SPLINE
SPL {X  -159.990, Y  +512.735, Z    +0.000, E1   +42.369, E3 +305939.523}
SPL {X  -159.990, Y  +505.924, Z    +0.000, E1   +43.199, E3 +305950.181}
SPL {X  -159.990, Y  +497.983, Z    +0.000, E1   +44.027, E3 +305963.054}
SPL {X  -159.990, Y  +489.703, Z    +0.000, E1   +44.938, E3 +305975.473}
SPL {X  -159.990, Y  +484.712, Z    +0.000, E1   +45.426, E3 +305983.087}
SPL {X  -159.990, Y  +477.648, Z    +0.000, E1   +46.080, E3 +305993.907}
SPL {X  -159.990, Y  +469.952, Z    +0.000, E1   +46.750, E3 +306005.415}
SPL {X  -159.990, Y  +462.892, Z    +0.000, E1   +47.497, E3 +306014.899}
SPL {X  -159.990, Y  +450.424, Z    +0.000, E1   +48.824, E3 +306030.863}
SPL {X  -159.990, Y  +436.919, Z    +0.000, E1   +49.944, E3 +306048.632}
SPL {X  -159.990, Y  +429.517, Z    +0.000, E1   +50.043, E3 +306061.146}
SPL {X  -159.990, Y  +423.834, Z    +0.000, E1   +50.037, E3 +306071.258}
SPL {X  -159.990, Y  +417.693, Z    +0.000, E1   +50.049, E3 +306082.156}
SPL {X  -159.990, Y  +408.922, Z    +0.000, E1   +50.085, E3 +306097.686}
SPL {X  -159.990, Y  +399.787, Z    +0.000, E1   +50.064, E3 +306113.955}
SPL {X  -159.990, Y  +393.038, Z    +0.000, E1   +50.038, E3 +306125.989}
SPL {X  -159.990, Y  +385.182, Z    +0.000, E1   +50.081, E3 +306139.906}
SPL {X  -159.906, Y  +377.302, Z    +0.000, E1   +50.024, E3 +306154.067}
SPL {X  -159.545, Y  +370.569, Z    +0.000, E1   +49.982, E3 +306166.380}
SPL {X  -158.871, Y  +363.614, Z    +0.000, E1   +49.855, E3 +306179.459}
SPL {X  -158.179, Y  +358.495, Z    +0.000, E1   +49.715, E3 +306189.308}
SPL {X  -157.354, Y  +353.576, Z    +0.000, E1   +49.583, E3 +306198.894}
SPL {X  -156.029, Y  +347.121, Z    +0.000, E1   +49.358, E3 +306211.711}
SPL {X  -154.686, Y  +341.646, Z    +0.000, E1   +49.094, E3 +306222.855}
SPL {X  -153.089, Y  +336.017, Z    +0.000, E1   +48.817, E3 +306234.464}
SPL {X  -151.481, Y  +331.019, Z    +0.000, E1   +48.491, E3 +306245.012}
SPL {X  -149.787, Y  +326.281, Z    +0.000, E1   +48.192, E3 +306255.100}
SPL {X  -148.124, Y  +322.035, Z    +0.000, E1   +47.846, E3 +306264.324}
SPL {X  -146.510, Y  +318.222, Z    +0.000, E1   +47.558, E3 +306272.636}
SPL {X  -141.189, Y  +307.250, Z    +0.000, E1   +40.067, E3 +306358.810}
ENDSPLINE

SPLINE
SPL {X  -154.923, Y  +342.556, Z    +0.000, E1   +23.930, E3 +306420.309}
SPL {X  -158.138, Y  +358.230, Z    +0.000, E1   +16.243, E3 +306429.267}
SPL {X  -159.647, Y  +372.034, Z    +0.000, E1    +8.739, E3 +306433.631}
SPL {X  -159.989, Y  +381.927, Z    +0.000, E1    +2.565, E3 +306435.391}
SPL {X  -159.990, Y  +386.909, Z    +0.000, E1    -1.211, E3 +306435.934}
SPL {X  -159.990, Y  +390.921, Z    +0.000, E1    -5.111, E3 +306436.413}
SPL {X  -159.990, Y  +395.719, Z    +0.000, E1   -10.396, E3 +306437.232}
SPL {X  -159.990, Y  +400.739, Z    +0.000, E1   -16.236, E3 +306438.430}
SPL {X  -159.990, Y  +409.482, Z    +0.000, E1   -25.418, E3 +306441.635}
SPL {X  -159.990, Y  +440.741, Z    +0.000, E1   -43.570, E3 +306462.292}
SPL {X  -159.990, Y  +489.732, Z    +0.000, E1   -48.863, E3 +306526.450}
SPL {X  -159.990, Y  +496.901, Z    +0.000, E1   -48.832, E3 +306539.797}
SPL {X  -159.990, Y  +502.531, Z    +0.000, E1   -48.834, E3 +306550.242}
SPL {X  -159.990, Y  +508.013, Z    +0.000, E1   -48.835, E3 +306560.377}
SPL {X  -159.990, Y  +513.813, Z    +0.000, E1   -48.843, E3 +306571.125}
SPL {X  -159.990, Y  +522.177, Z    +0.000, E1   -48.881, E3 +306586.602}
SPL {X  -159.990, Y  +532.076, Z    +0.000, E1   -48.872, E3 +306604.975}
SPL {X  -159.990, Y  +539.248, Z    +0.000, E1   -48.832, E3 +306618.343}
SPL {X  -159.990, Y  +544.926, Z    +0.000, E1   -48.835, E3 +306628.872}
SPL {X  -159.990, Y  +550.252, Z    +0.000, E1   -48.827, E3 +306638.778}
SPL {X  -159.990, Y  +555.692, Z    +0.000, E1   -48.830, E3 +306648.875}
SPL {X  -159.990, Y  +561.308, Z    +0.000, E1   -48.827, E3 +306659.322}
SPL {X  -159.990, Y  +566.669, Z    +0.000, E1   -48.820, E3 +306669.271}
SPL {X  -159.990, Y  +572.248, Z    +0.000, E1   -48.830, E3 +306679.616}
SPL {X  -159.990, Y  +577.770, Z    +0.000, E1   -48.821, E3 +306689.863}
SPL {X  -159.990, Y  +583.108, Z    +0.000, E1   -48.828, E3 +306699.765}
SPL {X  -159.990, Y  +588.804, Z    +0.000, E1   -48.829, E3 +306710.322}
SPL {X  -159.990, Y  +594.280, Z    +0.000, E1   -48.826, E3 +306720.484}
SPL {X  -159.990, Y  +600.107, Z    +0.000, E1   -48.833, E3 +306731.298}
SPL {X  -159.990, Y  +605.910, Z    +0.000, E1   -48.823, E3 +306742.077}
SPL {X  -159.990, Y  +611.566, Z    +0.000, E1   -48.829, E3 +306752.566}
SPL {X  -159.990, Y  +617.357, Z    +0.000, E1   -48.824, E3 +306763.321}
SPL {X  -159.990, Y  +622.965, Z    +0.000, E1   -48.826, E3 +306773.720}
SPL {X  -159.990, Y  +629.255, Z    +0.000, E1   -48.834, E3 +306785.387}
SPL {X  -159.990, Y  +634.905, Z    +0.000, E1   -48.821, E3 +306795.884}
SPL {X  -159.990, Y  +640.372, Z    +0.000, E1   -48.828, E3 +306806.021}
SPL {X  -159.990, Y  +646.939, Z    +0.000, E1   -48.838, E3 +306818.191}
SPL {X  -159.990, Y  +653.448, Z    +0.000, E1   -48.827, E3 +306830.286}
SPL {X  -159.990, Y  +659.039, Z    +0.000, E1   -48.826, E3 +306840.650}
SPL {X  -159.990, Y  +664.817, Z    +0.000, E1   -48.832, E3 +306851.365}
SPL {X  -159.990, Y  +671.221, Z    +0.000, E1   -48.836, E3 +306863.238}
SPL {X  -159.887, Y  +677.230, Z    +0.000, E1   -48.811, E3 +306874.504}
SPL {X  -159.602, Y  +682.629, Z    +0.000, E1   -48.761, E3 +306884.837}
SPL {X  -159.150, Y  +687.876, Z    +0.000, E1   -48.673, E3 +306895.076}
SPL {X  -158.569, Y  +692.776, Z    +0.000, E1   -48.570, E3 +306904.784}
SPL {X  -157.870, Y  +697.458, Z    +0.000, E1   -48.439, E3 +306914.213}
SPL {X  -157.028, Y  +702.144, Z    +0.000, E1   -48.297, E3 +306923.761}
SPL {X  -155.977, Y  +707.110, Z    +0.000, E1   -48.106, E3 +306934.065}
SPL {X  -154.657, Y  +712.464, Z    +0.000, E1   -47.874, E3 +306945.349}
SPL {X  -153.406, Y  +716.924, Z    +0.000, E1   -47.628, E3 +306954.915}
SPL {X  -152.020, Y  +721.367, Z    +0.000, E1   -47.374, E3 +306964.566}
SPL {X  -150.440, Y  +725.947, Z    +0.000, E1   -47.070, E3 +306974.671}
SPL {X  -148.730, Y  +730.459, Z    +0.000, E1   -46.749, E3 +306984.722}
SPL {X  -147.178, Y  +734.233, Z    +0.000, E1   -46.439, E3 +306993.256}
SPL {X  -140.222, Y  +748.536, Z    +0.000, E1   -42.074, E3 +307058.232}
ENDSPLINE

SPLINE
SPL {X  -152.021, Y  +721.365, Z    +0.000, E1   -28.339, E3 +307133.623}
SPL {X  -157.542, Y  +699.382, Z    +0.000, E1   -18.086, E3 +307149.141}
SPL {X  -159.386, Y  +685.393, Z    +0.000, E1   -10.664, E3 +307154.095}
SPL {X  -159.928, Y  +675.946, Z    +0.000, E1    -5.007, E3 +307156.134}
SPL {X  -159.990, Y  +671.468, Z    +0.000, E1    -2.030, E3 +307156.730}
SPL {X  -159.990, Y  +667.678, Z    +0.000, E1    +0.783, E3 +307157.080}
SPL {X  -159.990, Y  +663.139, Z    +0.000, E1    +5.135, E3 +307157.597}
SPL {X  -159.990, Y  +658.551, Z    +0.000, E1   +10.313, E3 +307158.371}
SPL {X  -159.990, Y  +653.526, Z    +0.000, E1   +16.156, E3 +307159.606}
SPL {X  -159.990, Y  +644.434, Z    +0.000, E1   +25.921, E3 +307162.801}
SPL {X  -159.990, Y  +612.255, Z    +0.000, E1   +44.102, E3 +307184.682}
SPL {X  -159.990, Y  +562.879, Z    +0.000, E1   +49.634, E3 +307246.271}
SPL {X  -159.990, Y  +554.544, Z    +0.000, E1   +49.649, E3 +307261.296}
SPL {X  -159.990, Y  +547.278, Z    +0.000, E1   +49.619, E3 +307274.455}
SPL {X  -159.990, Y  +540.489, Z    +0.000, E1   +49.634, E3 +307286.681}
SPL {X  -159.990, Y  +532.689, Z    +0.000, E1   +49.639, E3 +307300.734}
SPL {X  -159.990, Y  +524.316, Z    +0.000, E1   +49.648, E3 +307315.819}
SPL {X  -159.990, Y  +517.666, Z    +0.000, E1   +49.614, E3 +307327.880}
SPL {X  -159.990, Y  +511.038, Z    +0.000, E1   +49.636, E3 +307339.832}
SPL {X  -159.990, Y  +504.260, Z    +0.000, E1   +49.614, E3 +307352.105}
ENDSPLINE

SPLINE
SPL {X  -159.990, Y  +511.561, Z    +0.000, E1   +45.946, E3 +307359.627}
SPL {X  -159.990, Y  +518.175, Z    +0.000, E1   +41.708, E3 +307370.702}
ENDSPLINE

SPLINE
SPL {X  -159.990, Y  +508.096, Z    +0.000, E1   +42.952, E3 +307386.810}
SPL {X  -159.990, Y  +497.983, Z    +0.000, E1   +44.027, E3 +307403.054}
SPL {X  -159.990, Y  +489.703, Z    +0.000, E1   +44.938, E3 +307415.473}
SPL {X  -159.990, Y  +482.131, Z    +0.000, E1   +45.680, E3 +307427.053}
SPL {X  -159.990, Y  +472.111, Z    +0.000, E1   +46.581, E3 +307442.185}
SPL {X  -159.990, Y  +462.892, Z    +0.000, E1   +47.497, E3 +307454.899}
SPL {X  -159.990, Y  +452.841, Z    +0.000, E1   +48.572, E3 +307467.746}
SPL {X  -159.990, Y  +441.023, Z    +0.000, E1   +49.655, E3 +307482.997}
SPL {X  -159.990, Y  +431.096, Z    +0.000, E1   +50.075, E3 +307498.285}
SPL {X  -159.990, Y  +421.718, Z    +0.000, E1   +50.072, E3 +307514.965}
SPL {X  -159.990, Y  +412.896, Z    +0.000, E1   +50.065, E3 +307530.658}
SPL {X  -159.990, Y  +406.170, Z    +0.000, E1   +50.036, E3 +307542.647}
SPL {X  -159.990, Y  +399.787, Z    +0.000, E1   +50.064, E3 +307553.955}
SPL {X  -159.990, Y  +393.038, Z    +0.000, E1   +50.038, E3 +307565.989}
SPL {X  -159.990, Y  +385.182, Z    +0.000, E1   +50.081, E3 +307579.906}
SPL {X  -159.846, Y  +375.718, Z    +0.000, E1   +50.041, E3 +307596.901}
SPL {X  -159.300, Y  +367.653, Z    +0.000, E1   +49.944, E3 +307611.809}
SPL {X  -158.412, Y  +360.086, Z    +0.000, E1   +49.787, E3 +307626.191}
SPL {X  -157.354, Y  +353.576, Z    +0.000, E1   +49.583, E3 +307638.894}
SPL {X  -156.029, Y  +347.121, Z    +0.000, E1   +49.358, E3 +307651.711}
SPL {X  -154.686, Y  +341.646, Z    +0.000, E1   +49.094, E3 +307662.855}
SPL {X  -153.089, Y  +336.017, Z    +0.000, E1   +48.817, E3 +307674.464}
SPL {X  -151.481, Y  +331.019, Z    +0.000, E1   +48.491, E3 +307685.012}
SPL {X  -150.221, Y  +327.451, Z    +0.000, E1   +48.251, E3 +307692.616}
SPL {X  -148.587, Y  +323.181, Z    +0.000, E1   +47.960, E3 +307701.800}
SPL {X  -146.510, Y  +318.222, Z    +0.000, E1   +47.558, E3 +307712.636}
SPL {X  -141.189, Y  +307.250, Z    +0.000, E1   +40.067, E3 +307798.810}
ENDSPLINE

SPLINE
SPL {X  -154.923, Y  +342.556, Z    +0.000, E1   +23.930, E3 +307860.309}
SPL {X  -158.138, Y  +358.230, Z    +0.000, E1   +16.243, E3 +307869.267}
SPL {X  -159.647, Y  +372.034, Z    +0.000, E1    +8.739, E3 +307873.631}
SPL {X  -159.989, Y  +381.927, Z    +0.000, E1    +2.565, E3 +307875.391}
SPL {X  -159.990, Y  +386.909, Z    +0.000, E1    -1.211, E3 +307875.934}
SPL {X  -159.990, Y  +390.921, Z    +0.000, E1    -5.111, E3 +307876.413}
SPL {X  -159.990, Y  +395.719, Z    +0.000, E1   -10.396, E3 +307877.232}
SPL {X  -159.990, Y  +400.739, Z    +0.000, E1   -16.236, E3 +307878.430}
SPL {X  -159.990, Y  +409.482, Z    +0.000, E1   -25.418, E3 +307881.635}
SPL {X  -159.990, Y  +440.741, Z    +0.000, E1   -43.570, E3 +307902.292}
SPL {X  -159.990, Y  +488.072, Z    +0.000, E1   -48.834, E3 +307963.414}
SPL {X  -159.990, Y  +495.397, Z    +0.000, E1   -48.860, E3 +307976.963}
SPL {X  -159.990, Y  +502.531, Z    +0.000, E1   -48.834, E3 +307990.242}
SPL {X  -159.990, Y  +508.013, Z    +0.000, E1   -48.835, E3 +308000.377}
SPL {X  -159.990, Y  +513.813, Z    +0.000, E1   -48.843, E3 +308011.125}
SPL {X  -159.990, Y  +522.177, Z    +0.000, E1   -48.881, E3 +308026.602}
SPL {X  -159.990, Y  +532.076, Z    +0.000, E1   -48.872, E3 +308044.975}
SPL {X  -159.990, Y  +539.248, Z    +0.000, E1   -48.832, E3 +308058.343}
SPL {X  -159.990, Y  +544.926, Z    +0.000, E1   -48.835, E3 +308068.872}
SPL {X  -159.990, Y  +550.252, Z    +0.000, E1   -48.827, E3 +308078.778}
SPL {X  -159.990, Y  +555.692, Z    +0.000, E1   -48.830, E3 +308088.875}
SPL {X  -159.990, Y  +561.308, Z    +0.000, E1   -48.827, E3 +308099.322}
SPL {X  -159.990, Y  +566.669, Z    +0.000, E1   -48.820, E3 +308109.271}
SPL {X  -159.990, Y  +572.248, Z    +0.000, E1   -48.830, E3 +308119.616}
SPL {X  -159.990, Y  +577.770, Z    +0.000, E1   -48.821, E3 +308129.863}
SPL {X  -159.990, Y  +583.108, Z    +0.000, E1   -48.828, E3 +308139.765}
SPL {X  -159.990, Y  +588.804, Z    +0.000, E1   -48.829, E3 +308150.322}
SPL {X  -159.990, Y  +594.280, Z    +0.000, E1   -48.826, E3 +308160.484}
SPL {X  -159.990, Y  +600.107, Z    +0.000, E1   -48.833, E3 +308171.298}
SPL {X  -159.990, Y  +605.910, Z    +0.000, E1   -48.823, E3 +308182.077}
SPL {X  -159.990, Y  +611.566, Z    +0.000, E1   -48.829, E3 +308192.566}
SPL {X  -159.990, Y  +617.357, Z    +0.000, E1   -48.824, E3 +308203.321}
SPL {X  -159.990, Y  +622.965, Z    +0.000, E1   -48.826, E3 +308213.720}
SPL {X  -159.990, Y  +629.255, Z    +0.000, E1   -48.834, E3 +308225.387}
SPL {X  -159.990, Y  +634.905, Z    +0.000, E1   -48.821, E3 +308235.884}
SPL {X  -159.990, Y  +640.372, Z    +0.000, E1   -48.828, E3 +308246.021}
SPL {X  -159.990, Y  +646.939, Z    +0.000, E1   -48.838, E3 +308258.191}
SPL {X  -159.990, Y  +653.448, Z    +0.000, E1   -48.827, E3 +308270.286}
SPL {X  -159.990, Y  +659.039, Z    +0.000, E1   -48.826, E3 +308280.650}
SPL {X  -159.990, Y  +664.817, Z    +0.000, E1   -48.832, E3 +308291.365}
SPL {X  -159.990, Y  +671.221, Z    +0.000, E1   -48.836, E3 +308303.238}
SPL {X  -159.887, Y  +677.230, Z    +0.000, E1   -48.811, E3 +308314.504}
SPL {X  -159.602, Y  +682.629, Z    +0.000, E1   -48.761, E3 +308324.837}
SPL {X  -159.150, Y  +687.876, Z    +0.000, E1   -48.673, E3 +308335.076}
SPL {X  -158.569, Y  +692.776, Z    +0.000, E1   -48.570, E3 +308344.784}
SPL {X  -157.870, Y  +697.458, Z    +0.000, E1   -48.439, E3 +308354.213}
SPL {X  -157.028, Y  +702.144, Z    +0.000, E1   -48.297, E3 +308363.761}
SPL {X  -155.977, Y  +707.110, Z    +0.000, E1   -48.106, E3 +308374.065}
SPL {X  -154.657, Y  +712.464, Z    +0.000, E1   -47.874, E3 +308385.349}
SPL {X  -153.406, Y  +716.924, Z    +0.000, E1   -47.628, E3 +308394.915}
SPL {X  -152.020, Y  +721.367, Z    +0.000, E1   -47.374, E3 +308404.566}
SPL {X  -150.440, Y  +725.947, Z    +0.000, E1   -47.070, E3 +308414.671}
SPL {X  -148.730, Y  +730.459, Z    +0.000, E1   -46.749, E3 +308424.722}
SPL {X  -147.178, Y  +734.233, Z    +0.000, E1   -46.439, E3 +308433.256}
SPL {X  -140.263, Y  +748.461, Z    +0.000, E1   -42.675, E3 +308491.594}
ENDSPLINE

SPLINE
SPL {X  -141.835, Y  +745.525, Z    +0.000, E1   -39.068, E3 +308523.595}
SPL {X  -152.406, Y  +720.176, Z    +0.000, E1   -27.814, E3 +308574.808}
SPL {X  -158.165, Y  +695.595, Z    +0.000, E1   -16.189, E3 +308590.706}
SPL {X  -159.572, Y  +683.063, Z    +0.000, E1    -9.282, E3 +308594.713}
SPL {X  -159.928, Y  +675.946, Z    +0.000, E1    -5.007, E3 +308596.134}
SPL {X  -159.990, Y  +671.468, Z    +0.000, E1    -2.030, E3 +308596.730}
SPL {X  -159.990, Y  +667.678, Z    +0.000, E1    +0.783, E3 +308597.080}
SPL {X  -159.990, Y  +663.139, Z    +0.000, E1    +5.135, E3 +308597.597}
SPL {X  -159.990, Y  +658.551, Z    +0.000, E1   +10.313, E3 +308598.371}
SPL {X  -159.990, Y  +653.526, Z    +0.000, E1   +16.156, E3 +308599.606}
SPL {X  -159.990, Y  +644.434, Z    +0.000, E1   +25.921, E3 +308602.801}
SPL {X  -159.990, Y  +612.255, Z    +0.000, E1   +44.102, E3 +308624.682}
SPL {X  -159.990, Y  +567.037, Z    +0.000, E1   +49.607, E3 +308678.826}
SPL {X  -159.990, Y  +562.169, Z    +0.000, E1   +49.620, E3 +308687.582}
SPL {X  -159.990, Y  +554.544, Z    +0.000, E1   +49.649, E3 +308701.296}
SPL {X  -159.990, Y  +545.715, Z    +0.000, E1   +49.644, E3 +308717.240}
SPL {X  -159.990, Y  +537.339, Z    +0.000, E1   +49.638, E3 +308732.351}
SPL {X  -159.990, Y  +529.436, Z    +0.000, E1   +49.638, E3 +308746.603}
SPL {X  -159.990, Y  +520.280, Z    +0.000, E1   +49.665, E3 +308763.082}
SPL {X  -159.990, Y  +511.038, Z    +0.000, E1   +49.636, E3 +308779.832}
SPL {X  -159.990, Y  +504.260, Z    +0.000, E1   +49.614, E3 +308792.105}
ENDSPLINE

SPLINE
SPL {X  -159.990, Y  +511.561, Z    +0.000, E1   +45.946, E3 +308799.627}
SPL {X  -159.990, Y  +518.175, Z    +0.000, E1   +41.708, E3 +308810.702}
ENDSPLINE

SPLINE
SPL {X  -159.990, Y  +508.096, Z    +0.000, E1   +42.952, E3 +308826.810}
SPL {X  -159.990, Y  +497.983, Z    +0.000, E1   +44.027, E3 +308843.054}
SPL {X  -159.990, Y  +487.435, Z    +0.000, E1   +45.185, E3 +308858.910}
SPL {X  -159.990, Y  +477.648, Z    +0.000, E1   +46.080, E3 +308873.907}
SPL {X  -159.990, Y  +469.952, Z    +0.000, E1   +46.750, E3 +308885.415}
SPL {X  -159.990, Y  +462.892, Z    +0.000, E1   +47.497, E3 +308894.899}
SPL {X  -159.990, Y  +452.841, Z    +0.000, E1   +48.572, E3 +308907.746}
SPL {X  -159.990, Y  +439.038, Z    +0.000, E1   +49.804, E3 +308925.798}
SPL {X  -159.990, Y  +429.517, Z    +0.000, E1   +50.043, E3 +308941.146}
SPL {X  -159.990, Y  +423.834, Z    +0.000, E1   +50.037, E3 +308951.258}
SPL {X  -159.990, Y  +417.693, Z    +0.000, E1   +50.049, E3 +308962.156}
SPL {X  -159.990, Y  +411.447, Z    +0.000, E1   +50.039, E3 +308973.275}
SPL {X  -159.990, Y  +403.654, Z    +0.000, E1   +50.076, E3 +308987.065}
SPL {X  -159.990, Y  +394.612, Z    +0.000, E1   +50.064, E3 +309003.153}
SPL {X  -159.990, Y  +385.182, Z    +0.000, E1   +50.081, E3 +309019.906}
SPL {X  -159.846, Y  +375.718, Z    +0.000, E1   +50.041, E3 +309036.901}
SPL {X  -159.300, Y  +367.653, Z    +0.000, E1   +49.944, E3 +309051.809}
SPL {X  -158.412, Y  +360.086, Z    +0.000, E1   +49.787, E3 +309066.191}
SPL {X  -157.077, Y  +352.107, Z    +0.000, E1   +49.567, E3 +309081.742}
SPL {X  -155.744, Y  +345.884, Z    +0.000, E1   +49.283, E3 +309094.229}
SPL {X  -154.686, Y  +341.646, Z    +0.000, E1   +49.094, E3 +309102.855}
SPL {X  -153.089, Y  +336.017, Z    +0.000, E1   +48.817, E3 +309114.464}
SPL {X  -150.861, Y  +329.230, Z    +0.000, E1   +48.419, E3 +309128.753}
SPL {X  -148.587, Y  +323.181, Z    +0.000, E1   +47.960, E3 +309141.800}
SPL {X  -146.885, Y  +319.085, Z    +0.000, E1   +47.613, E3 +309150.761}
SPL {X  -145.797, Y  +316.621, Z    +0.000, E1   +47.387, E3 +309156.210}
SPL {X  -141.189, Y  +307.250, Z    +0.000, E1   +40.067, E3 +309238.810}
ENDSPLINE

SPLINE
SPL {X  -154.923, Y  +342.556, Z    +0.000, E1   +23.930, E3 +309300.309}
SPL {X  -158.138, Y  +358.230, Z    +0.000, E1   +16.243, E3 +309309.267}
SPL {X  -159.407, Y  +368.849, Z    +0.000, E1   +10.504, E3 +309312.867}
SPL {X  -159.931, Y  +378.162, Z    +0.000, E1    +5.020, E3 +309314.852}
SPL {X  -159.990, Y  +383.297, Z    +0.000, E1    +1.526, E3 +309315.557}
SPL {X  -159.990, Y  +386.909, Z    +0.000, E1    -1.211, E3 +309315.934}
SPL {X  -159.990, Y  +390.921, Z    +0.000, E1    -5.111, E3 +309316.413}
SPL {X  -159.990, Y  +395.719, Z    +0.000, E1   -10.396, E3 +309317.232}
SPL {X  -159.990, Y  +400.739, Z    +0.000, E1   -16.236, E3 +309318.430}
SPL {X  -159.990, Y  +409.482, Z    +0.000, E1   -25.418, E3 +309321.635}
SPL {X  -159.990, Y  +440.741, Z    +0.000, E1   -43.570, E3 +309342.292}
SPL {X  -159.990, Y  +489.732, Z    +0.000, E1   -48.863, E3 +309406.450}
SPL {X  -159.990, Y  +496.901, Z    +0.000, E1   -48.832, E3 +309419.797}
SPL {X  -159.990, Y  +502.531, Z    +0.000, E1   -48.834, E3 +309430.242}
SPL {X  -159.990, Y  +508.013, Z    +0.000, E1   -48.835, E3 +309440.377}
SPL {X  -159.990, Y  +513.813, Z    +0.000, E1   -48.843, E3 +309451.125}
SPL {X  -159.990, Y  +522.177, Z    +0.000, E1   -48.881, E3 +309466.602}
SPL {X  -159.990, Y  +532.076, Z    +0.000, E1   -48.872, E3 +309484.975}
SPL {X  -159.990, Y  +539.248, Z    +0.000, E1   -48.832, E3 +309498.343}
SPL {X  -159.990, Y  +544.926, Z    +0.000, E1   -48.835, E3 +309508.872}
SPL {X  -159.990, Y  +550.252, Z    +0.000, E1   -48.827, E3 +309518.778}
SPL {X  -159.990, Y  +555.692, Z    +0.000, E1   -48.830, E3 +309528.875}
SPL {X  -159.990, Y  +561.308, Z    +0.000, E1   -48.827, E3 +309539.322}
SPL {X  -159.990, Y  +566.669, Z    +0.000, E1   -48.820, E3 +309549.271}
SPL {X  -159.990, Y  +572.248, Z    +0.000, E1   -48.830, E3 +309559.616}
SPL {X  -159.990, Y  +577.770, Z    +0.000, E1   -48.821, E3 +309569.863}
SPL {X  -159.990, Y  +583.108, Z    +0.000, E1   -48.828, E3 +309579.765}
SPL {X  -159.990, Y  +588.804, Z    +0.000, E1   -48.829, E3 +309590.322}
SPL {X  -159.990, Y  +594.280, Z    +0.000, E1   -48.826, E3 +309600.484}
SPL {X  -159.990, Y  +600.107, Z    +0.000, E1   -48.833, E3 +309611.298}
SPL {X  -159.990, Y  +605.910, Z    +0.000, E1   -48.823, E3 +309622.077}
SPL {X  -159.990, Y  +611.566, Z    +0.000, E1   -48.829, E3 +309632.566}
SPL {X  -159.990, Y  +617.357, Z    +0.000, E1   -48.824, E3 +309643.321}
SPL {X  -159.990, Y  +622.965, Z    +0.000, E1   -48.826, E3 +309653.720}
SPL {X  -159.990, Y  +629.255, Z    +0.000, E1   -48.834, E3 +309665.387}
SPL {X  -159.990, Y  +634.905, Z    +0.000, E1   -48.821, E3 +309675.884}
SPL {X  -159.990, Y  +640.372, Z    +0.000, E1   -48.828, E3 +309686.021}
SPL {X  -159.990, Y  +646.939, Z    +0.000, E1   -48.838, E3 +309698.191}
SPL {X  -159.990, Y  +653.448, Z    +0.000, E1   -48.827, E3 +309710.286}
SPL {X  -159.990, Y  +659.039, Z    +0.000, E1   -48.826, E3 +309720.650}
SPL {X  -159.990, Y  +664.817, Z    +0.000, E1   -48.832, E3 +309731.365}
SPL {X  -159.990, Y  +671.221, Z    +0.000, E1   -48.836, E3 +309743.238}
SPL {X  -159.887, Y  +677.230, Z    +0.000, E1   -48.811, E3 +309754.504}
SPL {X  -159.602, Y  +682.629, Z    +0.000, E1   -48.761, E3 +309764.837}
SPL {X  -159.150, Y  +687.876, Z    +0.000, E1   -48.673, E3 +309775.076}
SPL {X  -158.569, Y  +692.776, Z    +0.000, E1   -48.570, E3 +309784.784}
SPL {X  -157.870, Y  +697.458, Z    +0.000, E1   -48.439, E3 +309794.213}
SPL {X  -157.028, Y  +702.144, Z    +0.000, E1   -48.297, E3 +309803.761}
SPL {X  -155.977, Y  +707.110, Z    +0.000, E1   -48.106, E3 +309814.065}
SPL {X  -154.657, Y  +712.464, Z    +0.000, E1   -47.874, E3 +309825.349}
SPL {X  -153.406, Y  +716.924, Z    +0.000, E1   -47.628, E3 +309834.915}
SPL {X  -152.020, Y  +721.367, Z    +0.000, E1   -47.374, E3 +309844.566}
SPL {X  -150.440, Y  +725.947, Z    +0.000, E1   -47.070, E3 +309854.671}
SPL {X  -148.730, Y  +730.459, Z    +0.000, E1   -46.749, E3 +309864.722}
SPL {X  -147.178, Y  +734.233, Z    +0.000, E1   -46.439, E3 +309873.256}
SPL {X  -140.222, Y  +748.536, Z    +0.000, E1   -42.074, E3 +309938.232}
ENDSPLINE

SPLINE
SPL {X  -152.021, Y  +721.365, Z    +0.000, E1   -28.339, E3 +310013.623}
SPL {X  -158.165, Y  +695.595, Z    +0.000, E1   -16.189, E3 +310030.706}
SPL {X  -159.572, Y  +683.063, Z    +0.000, E1    -9.282, E3 +310034.713}
SPL {X  -159.928, Y  +675.946, Z    +0.000, E1    -5.007, E3 +310036.134}
SPL {X  -159.990, Y  +669.697, Z    +0.000, E1    -0.851, E3 +310036.894}
SPL {X  -159.990, Y  +665.698, Z    +0.000, E1    +2.616, E3 +310037.273}
SPL {X  -159.990, Y  +662.251, Z    +0.000, E1    +6.155, E3 +310037.719}
SPL {X  -159.990, Y  +658.551, Z    +0.000, E1   +10.313, E3 +310038.371}
SPL {X  -159.990, Y  +653.526, Z    +0.000, E1   +16.156, E3 +310039.606}
SPL {X  -159.990, Y  +644.434, Z    +0.000, E1   +25.921, E3 +310042.801}
SPL {X  -159.990, Y  +612.255, Z    +0.000, E1   +44.102, E3 +310064.682}
SPL {X  -159.990, Y  +561.053, Z    +0.000, E1   +49.668, E3 +310129.515}
SPL {X  -159.990, Y  +552.984, Z    +0.000, E1   +49.619, E3 +310144.156}
SPL {X  -159.990, Y  +547.278, Z    +0.000, E1   +49.619, E3 +310154.455}
SPL {X  -159.990, Y  +538.738, Z    +0.000, E1   +49.672, E3 +310169.779}
SPL {X  -159.990, Y  +529.436, Z    +0.000, E1   +49.638, E3 +310186.603}
SPL {X  -159.990, Y  +522.804, Z    +0.000, E1   +49.620, E3 +310198.592}
SPL {X  -159.990, Y  +515.173, Z    +0.000, E1   +49.653, E3 +310212.330}
SPL {X  -159.990, Y  +505.472, Z    +0.000, E1   +49.465, E3 +310231.135}
ENDSPLINE

SPLINE
SPL {X  -159.990, Y  +518.841, Z    +0.000, E1   +41.643, E3 +310249.543}
ENDSPLINE

SPLINE
SPL {X  -159.990, Y  +508.096, Z    +0.000, E1   +42.952, E3 +310266.810}
SPL {X  -159.990, Y  +500.642, Z    +0.000, E1   +43.747, E3 +310278.731}
SPL {X  -159.990, Y  +495.820, Z    +0.000, E1   +44.207, E3 +310286.618}
SPL {X  -159.990, Y  +487.435, Z    +0.000, E1   +45.185, E3 +310298.910}
SPL {X  -159.990, Y  +477.648, Z    +0.000, E1   +46.080, E3 +310313.907}
SPL {X  -159.990, Y  +469.952, Z    +0.000, E1   +46.750, E3 +310325.415}
SPL {X  -159.990, Y  +462.892, Z    +0.000, E1   +47.497, E3 +310334.899}
SPL {X  -159.990, Y  +452.841, Z    +0.000, E1   +48.572, E3 +310347.746}
SPL {X  -159.990, Y  +439.038, Z    +0.000, E1   +49.804, E3 +310365.798}
SPL {X  -159.990, Y  +429.517, Z    +0.000, E1   +50.043, E3 +310381.146}
SPL {X  -159.990, Y  +423.834, Z    +0.000, E1   +50.037, E3 +310391.258}
SPL {X  -159.990, Y  +417.693, Z    +0.000, E1   +50.049, E3 +310402.156}
SPL {X  -159.990, Y  +411.447, Z    +0.000, E1   +50.039, E3 +310413.275}
SPL {X  -159.990, Y  +406.170, Z    +0.000, E1   +50.036, E3 +310422.647}
SPL {X  -159.990, Y  +399.787, Z    +0.000, E1   +50.064, E3 +310433.955}
SPL {X  -159.990, Y  +393.038, Z    +0.000, E1   +50.038, E3 +310445.989}
SPL {X  -159.990, Y  +387.356, Z    +0.000, E1   +50.042, E3 +310456.100}
SPL {X  -159.990, Y  +382.225, Z    +0.000, E1   +50.028, E3 +310465.245}
SPL {X  -159.846, Y  +375.718, Z    +0.000, E1   +50.041, E3 +310476.901}
SPL {X  -159.443, Y  +369.277, Z    +0.000, E1   +49.941, E3 +310488.815}
SPL {X  -158.871, Y  +363.614, Z    +0.000, E1   +49.855, E3 +310499.459}
SPL {X  -158.179, Y  +358.495, Z    +0.000, E1   +49.715, E3 +310509.308}
SPL {X  -157.077, Y  +352.107, Z    +0.000, E1   +49.567, E3 +310521.742}
SPL {X  -155.744, Y  +345.884, Z    +0.000, E1   +49.283, E3 +310534.229}
SPL {X  -154.686, Y  +341.646, Z    +0.000, E1   +49.094, E3 +310542.855}
SPL {X  -153.439, Y  +337.188, Z    +0.000, E1   +48.857, E3 +310552.062}
SPL {X  -151.836, Y  +332.074, Z    +0.000, E1   +48.585, E3 +310562.738}
SPL {X  -150.221, Y  +327.451, Z    +0.000, E1   +48.251, E3 +310572.616}
SPL {X  -148.587, Y  +323.181, Z    +0.000, E1   +47.960, E3 +310581.800}
SPL {X  -146.510, Y  +318.222, Z    +0.000, E1   +47.558, E3 +310592.636}
SPL {X  -141.189, Y  +307.250, Z    +0.000, E1   +40.067, E3 +310678.810}
ENDSPLINE

SPLINE
SPL {X  -154.923, Y  +342.556, Z    +0.000, E1   +23.930, E3 +310740.309}
SPL {X  -158.138, Y  +358.230, Z    +0.000, E1   +16.243, E3 +310749.267}
SPL {X  -159.647, Y  +372.034, Z    +0.000, E1    +8.739, E3 +310753.631}
SPL {X  -159.989, Y  +381.927, Z    +0.000, E1    +2.565, E3 +310755.391}
SPL {X  -159.990, Y  +386.909, Z    +0.000, E1    -1.211, E3 +310755.934}
SPL {X  -159.990, Y  +390.921, Z    +0.000, E1    -5.111, E3 +310756.413}
SPL {X  -159.990, Y  +395.719, Z    +0.000, E1   -10.396, E3 +310757.232}
SPL {X  -159.990, Y  +400.739, Z    +0.000, E1   -16.236, E3 +310758.430}
SPL {X  -159.990, Y  +409.482, Z    +0.000, E1   -25.418, E3 +310761.635}
SPL {X  -159.990, Y  +440.741, Z    +0.000, E1   -43.570, E3 +310782.292}
SPL {X  -159.990, Y  +489.732, Z    +0.000, E1   -48.863, E3 +310846.450}
SPL {X  -159.990, Y  +496.901, Z    +0.000, E1   -48.832, E3 +310859.797}
SPL {X  -159.990, Y  +502.531, Z    +0.000, E1   -48.834, E3 +310870.242}
SPL {X  -159.990, Y  +508.013, Z    +0.000, E1   -48.835, E3 +310880.377}
SPL {X  -159.990, Y  +513.813, Z    +0.000, E1   -48.843, E3 +310891.125}
SPL {X  -159.990, Y  +522.177, Z    +0.000, E1   -48.881, E3 +310906.602}
SPL {X  -159.990, Y  +532.076, Z    +0.000, E1   -48.872, E3 +310924.975}
SPL {X  -159.990, Y  +539.248, Z    +0.000, E1   -48.832, E3 +310938.343}
SPL {X  -159.990, Y  +544.926, Z    +0.000, E1   -48.835, E3 +310948.872}
SPL {X  -159.990, Y  +550.252, Z    +0.000, E1   -48.827, E3 +310958.778}
SPL {X  -159.990, Y  +555.692, Z    +0.000, E1   -48.830, E3 +310968.875}
SPL {X  -159.990, Y  +561.308, Z    +0.000, E1   -48.827, E3 +310979.322}
SPL {X  -159.990, Y  +566.669, Z    +0.000, E1   -48.820, E3 +310989.271}
SPL {X  -159.990, Y  +572.248, Z    +0.000, E1   -48.830, E3 +310999.616}
SPL {X  -159.990, Y  +577.770, Z    +0.000, E1   -48.821, E3 +311009.863}
SPL {X  -159.990, Y  +583.108, Z    +0.000, E1   -48.828, E3 +311019.765}
SPL {X  -159.990, Y  +588.804, Z    +0.000, E1   -48.829, E3 +311030.322}
SPL {X  -159.990, Y  +594.280, Z    +0.000, E1   -48.826, E3 +311040.484}
SPL {X  -159.990, Y  +600.107, Z    +0.000, E1   -48.833, E3 +311051.298}
SPL {X  -159.990, Y  +605.910, Z    +0.000, E1   -48.823, E3 +311062.077}
SPL {X  -159.990, Y  +611.566, Z    +0.000, E1   -48.829, E3 +311072.566}
SPL {X  -159.990, Y  +617.357, Z    +0.000, E1   -48.824, E3 +311083.321}
SPL {X  -159.990, Y  +622.965, Z    +0.000, E1   -48.826, E3 +311093.720}
SPL {X  -159.990, Y  +629.255, Z    +0.000, E1   -48.834, E3 +311105.387}
SPL {X  -159.990, Y  +634.905, Z    +0.000, E1   -48.821, E3 +311115.884}
SPL {X  -159.990, Y  +640.372, Z    +0.000, E1   -48.828, E3 +311126.021}
SPL {X  -159.990, Y  +646.939, Z    +0.000, E1   -48.838, E3 +311138.191}
SPL {X  -159.990, Y  +653.448, Z    +0.000, E1   -48.827, E3 +311150.286}
SPL {X  -159.990, Y  +659.039, Z    +0.000, E1   -48.826, E3 +311160.650}
SPL {X  -159.990, Y  +664.817, Z    +0.000, E1   -48.832, E3 +311171.365}
SPL {X  -159.990, Y  +671.221, Z    +0.000, E1   -48.836, E3 +311183.238}
SPL {X  -159.887, Y  +677.230, Z    +0.000, E1   -48.811, E3 +311194.504}
SPL {X  -159.602, Y  +682.629, Z    +0.000, E1   -48.761, E3 +311204.837}
SPL {X  -159.150, Y  +687.876, Z    +0.000, E1   -48.673, E3 +311215.076}
SPL {X  -158.569, Y  +692.776, Z    +0.000, E1   -48.570, E3 +311224.784}
SPL {X  -157.870, Y  +697.458, Z    +0.000, E1   -48.439, E3 +311234.213}
SPL {X  -157.028, Y  +702.144, Z    +0.000, E1   -48.297, E3 +311243.761}
SPL {X  -155.977, Y  +707.110, Z    +0.000, E1   -48.106, E3 +311254.065}
SPL {X  -154.657, Y  +712.464, Z    +0.000, E1   -47.874, E3 +311265.349}
SPL {X  -153.406, Y  +716.924, Z    +0.000, E1   -47.628, E3 +311274.915}
SPL {X  -152.020, Y  +721.367, Z    +0.000, E1   -47.374, E3 +311284.566}
SPL {X  -150.440, Y  +725.947, Z    +0.000, E1   -47.070, E3 +311294.671}
SPL {X  -148.730, Y  +730.459, Z    +0.000, E1   -46.749, E3 +311304.722}
SPL {X  -147.178, Y  +734.233, Z    +0.000, E1   -46.439, E3 +311313.256}
SPL {X  -140.263, Y  +748.461, Z    +0.000, E1   -42.675, E3 +311371.594}
ENDSPLINE

SPLINE
SPL {X  -141.835, Y  +745.525, Z    +0.000, E1   -39.068, E3 +311403.595}
SPL {X  -152.406, Y  +720.176, Z    +0.000, E1   -27.814, E3 +311454.808}
SPL {X  -157.542, Y  +699.382, Z    +0.000, E1   -18.086, E3 +311469.141}
SPL {X  -159.386, Y  +685.393, Z    +0.000, E1   -10.664, E3 +311474.095}
SPL {X  -159.928, Y  +675.946, Z    +0.000, E1    -5.007, E3 +311476.134}
SPL {X  -159.990, Y  +671.468, Z    +0.000, E1    -2.030, E3 +311476.730}
SPL {X  -159.990, Y  +667.678, Z    +0.000, E1    +0.783, E3 +311477.080}
SPL {X  -159.990, Y  +663.139, Z    +0.000, E1    +5.135, E3 +311477.597}
SPL {X  -159.990, Y  +658.551, Z    +0.000, E1   +10.313, E3 +311478.371}
SPL {X  -159.990, Y  +653.526, Z    +0.000, E1   +16.156, E3 +311479.606}
SPL {X  -159.990, Y  +644.434, Z    +0.000, E1   +25.921, E3 +311482.801}
SPL {X  -159.990, Y  +612.255, Z    +0.000, E1   +44.102, E3 +311504.682}
SPL {X  -159.990, Y  +561.053, Z    +0.000, E1   +49.668, E3 +311569.515}
SPL {X  -159.990, Y  +552.984, Z    +0.000, E1   +49.619, E3 +311584.156}
SPL {X  -159.990, Y  +547.278, Z    +0.000, E1   +49.619, E3 +311594.455}
SPL {X  -159.990, Y  +538.738, Z    +0.000, E1   +49.672, E3 +311609.779}
SPL {X  -159.990, Y  +529.436, Z    +0.000, E1   +49.638, E3 +311626.603}
SPL {X  -159.990, Y  +520.280, Z    +0.000, E1   +49.665, E3 +311643.082}
SPL {X  -159.990, Y  +511.038, Z    +0.000, E1   +49.636, E3 +311659.832}
SPL {X  -159.990, Y  +504.260, Z    +0.000, E1   +49.614, E3 +311672.105}
SPL {X  -159.990, Y  +503.881, Z    +0.000, E1   +48.376, E3 +311680.092}
ENDSPLINE

SPLINE
SPL {X  -159.990, Y  +520.622, Z    +0.000, E1   +41.395, E3 +311686.672}
ENDSPLINE

SPLINE
SPL {X  -159.990, Y  +512.735, Z    +0.000, E1   +42.369, E3 +311699.523}
SPL {X  -159.990, Y  +505.924, Z    +0.000, E1   +43.199, E3 +311710.181}
SPL {X  -159.990, Y  +497.983, Z    +0.000, E1   +44.027, E3 +311723.054}
SPL {X  -159.990, Y  +489.703, Z    +0.000, E1   +44.938, E3 +311735.473}
SPL {X  -159.990, Y  +484.712, Z    +0.000, E1   +45.426, E3 +311743.087}
SPL {X  -159.990, Y  +477.648, Z    +0.000, E1   +46.080, E3 +311753.907}
SPL {X  -159.990, Y  +469.952, Z    +0.000, E1   +46.750, E3 +311765.415}
SPL {X  -159.990, Y  +462.892, Z    +0.000, E1   +47.497, E3 +311774.899}
SPL {X  -159.990, Y  +450.424, Z    +0.000, E1   +48.824, E3 +311790.863}
SPL {X  -159.990, Y  +436.919, Z    +0.000, E1   +49.944, E3 +311808.632}
SPL {X  -159.990, Y  +429.517, Z    +0.000, E1   +50.043, E3 +311821.146}
SPL {X  -159.990, Y  +423.834, Z    +0.000, E1   +50.037, E3 +311831.258}
SPL {X  -159.990, Y  +417.693, Z    +0.000, E1   +50.049, E3 +311842.156}
SPL {X  -159.990, Y  +408.922, Z    +0.000, E1   +50.085, E3 +311857.686}
SPL {X  -159.990, Y  +399.787, Z    +0.000, E1   +50.064, E3 +311873.955}
SPL {X  -159.990, Y  +393.038, Z    +0.000, E1   +50.038, E3 +311885.989}
SPL {X  -159.990, Y  +385.182, Z    +0.000, E1   +50.081, E3 +311899.906}
SPL {X  -159.906, Y  +377.302, Z    +0.000, E1   +50.024, E3 +311914.067}
SPL {X  -159.545, Y  +370.569, Z    +0.000, E1   +49.982, E3 +311926.380}
SPL {X  -158.871, Y  +363.614, Z    +0.000, E1   +49.855, E3 +311939.459}
SPL {X  -158.179, Y  +358.495, Z    +0.000, E1   +49.715, E3 +311949.308}
SPL {X  -157.354, Y  +353.576, Z    +0.000, E1   +49.583, E3 +311958.894}
SPL {X  -156.029, Y  +347.121, Z    +0.000, E1   +49.358, E3 +311971.711}
SPL {X  -154.686, Y  +341.646, Z    +0.000, E1   +49.094, E3 +311982.855}
SPL {X  -153.089, Y  +336.017, Z    +0.000, E1   +48.817, E3 +311994.464}
SPL {X  -151.481, Y  +331.019, Z    +0.000, E1   +48.491, E3 +312005.012}
SPL {X  -149.787, Y  +326.281, Z    +0.000, E1   +48.192, E3 +312015.100}
SPL {X  -148.124, Y  +322.035, Z    +0.000, E1   +47.846, E3 +312024.324}
SPL {X  -146.510, Y  +318.222, Z    +0.000, E1   +47.558, E3 +312032.636}
SPL {X  -141.189, Y  +307.250, Z    +0.000, E1   +40.067, E3 +312118.810}
ENDSPLINE

SPLINE
SPL {X  -154.923, Y  +342.556, Z    +0.000, E1   +23.930, E3 +312180.309}
SPL {X  -158.138, Y  +358.230, Z    +0.000, E1   +16.243, E3 +312189.267}
SPL {X  -159.407, Y  +368.849, Z    +0.000, E1   +10.504, E3 +312192.867}
SPL {X  -159.931, Y  +378.162, Z    +0.000, E1    +5.020, E3 +312194.852}
SPL {X  -159.990, Y  +383.297, Z    +0.000, E1    +1.526, E3 +312195.557}
SPL {X  -159.990, Y  +386.909, Z    +0.000, E1    -1.211, E3 +312195.934}
SPL {X  -159.990, Y  +390.921, Z    +0.000, E1    -5.111, E3 +312196.413}
SPL {X  -159.990, Y  +395.719, Z    +0.000, E1   -10.396, E3 +312197.232}
SPL {X  -159.990, Y  +400.739, Z    +0.000, E1   -16.236, E3 +312198.430}
SPL {X  -159.990, Y  +409.482, Z    +0.000, E1   -25.418, E3 +312201.635}
SPL {X  -159.990, Y  +440.741, Z    +0.000, E1   -43.570, E3 +312222.292}
SPL {X  -159.990, Y  +489.732, Z    +0.000, E1   -48.863, E3 +312286.450}
SPL {X  -159.990, Y  +496.901, Z    +0.000, E1   -48.832, E3 +312299.797}
SPL {X  -159.990, Y  +502.531, Z    +0.000, E1   -48.834, E3 +312310.242}
SPL {X  -159.990, Y  +508.013, Z    +0.000, E1   -48.835, E3 +312320.377}
SPL {X  -159.990, Y  +513.813, Z    +0.000, E1   -48.843, E3 +312331.125}
SPL {X  -159.990, Y  +522.177, Z    +0.000, E1   -48.881, E3 +312346.602}
SPL {X  -159.990, Y  +532.076, Z    +0.000, E1   -48.872, E3 +312364.975}
SPL {X  -159.990, Y  +539.248, Z    +0.000, E1   -48.832, E3 +312378.343}
SPL {X  -159.990, Y  +544.926, Z    +0.000, E1   -48.835, E3 +312388.872}
SPL {X  -159.990, Y  +550.252, Z    +0.000, E1   -48.827, E3 +312398.778}
SPL {X  -159.990, Y  +555.692, Z    +0.000, E1   -48.830, E3 +312408.875}
SPL {X  -159.990, Y  +561.308, Z    +0.000, E1   -48.827, E3 +312419.322}
SPL {X  -159.990, Y  +566.669, Z    +0.000, E1   -48.820, E3 +312429.271}
SPL {X  -159.990, Y  +572.248, Z    +0.000, E1   -48.830, E3 +312439.616}
SPL {X  -159.990, Y  +577.770, Z    +0.000, E1   -48.821, E3 +312449.863}
SPL {X  -159.990, Y  +583.108, Z    +0.000, E1   -48.828, E3 +312459.765}
SPL {X  -159.990, Y  +588.804, Z    +0.000, E1   -48.829, E3 +312470.322}
SPL {X  -159.990, Y  +594.280, Z    +0.000, E1   -48.826, E3 +312480.484}
SPL {X  -159.990, Y  +600.107, Z    +0.000, E1   -48.833, E3 +312491.298}
SPL {X  -159.990, Y  +605.910, Z    +0.000, E1   -48.823, E3 +312502.077}
SPL {X  -159.990, Y  +611.566, Z    +0.000, E1   -48.829, E3 +312512.566}
SPL {X  -159.990, Y  +617.357, Z    +0.000, E1   -48.824, E3 +312523.321}
SPL {X  -159.990, Y  +622.965, Z    +0.000, E1   -48.826, E3 +312533.720}
SPL {X  -159.990, Y  +629.255, Z    +0.000, E1   -48.834, E3 +312545.387}
SPL {X  -159.990, Y  +634.905, Z    +0.000, E1   -48.821, E3 +312555.884}
SPL {X  -159.990, Y  +640.372, Z    +0.000, E1   -48.828, E3 +312566.021}
SPL {X  -159.990, Y  +646.939, Z    +0.000, E1   -48.838, E3 +312578.191}
SPL {X  -159.990, Y  +653.448, Z    +0.000, E1   -48.827, E3 +312590.286}
SPL {X  -159.990, Y  +659.039, Z    +0.000, E1   -48.826, E3 +312600.650}
SPL {X  -159.990, Y  +664.817, Z    +0.000, E1   -48.832, E3 +312611.365}
SPL {X  -159.990, Y  +671.221, Z    +0.000, E1   -48.836, E3 +312623.238}
SPL {X  -159.887, Y  +677.230, Z    +0.000, E1   -48.811, E3 +312634.504}
SPL {X  -159.602, Y  +682.629, Z    +0.000, E1   -48.761, E3 +312644.837}
SPL {X  -159.150, Y  +687.876, Z    +0.000, E1   -48.673, E3 +312655.076}
SPL {X  -158.569, Y  +692.776, Z    +0.000, E1   -48.570, E3 +312664.784}
SPL {X  -157.870, Y  +697.458, Z    +0.000, E1   -48.439, E3 +312674.213}
SPL {X  -157.028, Y  +702.144, Z    +0.000, E1   -48.297, E3 +312683.761}
SPL {X  -155.977, Y  +707.110, Z    +0.000, E1   -48.106, E3 +312694.065}
SPL {X  -154.657, Y  +712.464, Z    +0.000, E1   -47.874, E3 +312705.349}
SPL {X  -153.406, Y  +716.924, Z    +0.000, E1   -47.628, E3 +312714.915}
SPL {X  -152.020, Y  +721.367, Z    +0.000, E1   -47.374, E3 +312724.566}
SPL {X  -150.440, Y  +725.947, Z    +0.000, E1   -47.070, E3 +312734.671}
SPL {X  -148.730, Y  +730.459, Z    +0.000, E1   -46.749, E3 +312744.722}
SPL {X  -147.178, Y  +734.233, Z    +0.000, E1   -46.439, E3 +312753.256}
SPL {X  -140.222, Y  +748.536, Z    +0.000, E1   -42.074, E3 +312818.232}
ENDSPLINE

SPLINE
SPL {X  -152.021, Y  +721.365, Z    +0.000, E1   -28.339, E3 +312893.623}
SPL {X  -158.165, Y  +695.595, Z    +0.000, E1   -16.189, E3 +312910.706}
SPL {X  -159.572, Y  +683.063, Z    +0.000, E1    -9.282, E3 +312914.713}
SPL {X  -159.928, Y  +675.946, Z    +0.000, E1    -5.007, E3 +312916.134}
SPL {X  -159.990, Y  +669.697, Z    +0.000, E1    -0.851, E3 +312916.894}
SPL {X  -159.990, Y  +665.698, Z    +0.000, E1    +2.616, E3 +312917.273}
SPL {X  -159.990, Y  +662.251, Z    +0.000, E1    +6.155, E3 +312917.719}
SPL {X  -159.990, Y  +658.551, Z    +0.000, E1   +10.313, E3 +312918.371}
SPL {X  -159.990, Y  +653.526, Z    +0.000, E1   +16.156, E3 +312919.606}
SPL {X  -159.990, Y  +644.434, Z    +0.000, E1   +25.921, E3 +312922.801}
SPL {X  -159.990, Y  +612.255, Z    +0.000, E1   +44.102, E3 +312944.682}
SPL {X  -159.990, Y  +561.053, Z    +0.000, E1   +49.668, E3 +313009.515}
SPL {X  -159.990, Y  +552.984, Z    +0.000, E1   +49.619, E3 +313024.156}
SPL {X  -159.990, Y  +547.278, Z    +0.000, E1   +49.619, E3 +313034.455}
SPL {X  -159.990, Y  +538.738, Z    +0.000, E1   +49.672, E3 +313049.779}
SPL {X  -159.990, Y  +529.436, Z    +0.000, E1   +49.638, E3 +313066.603}
SPL {X  -159.990, Y  +522.804, Z    +0.000, E1   +49.620, E3 +313078.592}
SPL {X  -159.990, Y  +515.173, Z    +0.000, E1   +49.653, E3 +313092.330}
SPL {X  -159.990, Y  +505.472, Z    +0.000, E1   +49.465, E3 +313111.135}
ENDSPLINE

SPLINE
SPL {X  -159.990, Y  +518.841, Z    +0.000, E1   +41.643, E3 +313129.543}
ENDSPLINE

SPLINE
SPL {X  -159.990, Y  +508.096, Z    +0.000, E1   +42.952, E3 +313146.810}
SPL {X  -159.990, Y  +500.642, Z    +0.000, E1   +43.747, E3 +313158.731}
SPL {X  -159.990, Y  +495.820, Z    +0.000, E1   +44.207, E3 +313166.618}
SPL {X  -159.990, Y  +487.435, Z    +0.000, E1   +45.185, E3 +313178.910}
SPL {X  -159.990, Y  +477.648, Z    +0.000, E1   +46.080, E3 +313193.907}
SPL {X  -159.990, Y  +469.952, Z    +0.000, E1   +46.750, E3 +313205.415}
SPL {X  -159.990, Y  +462.892, Z    +0.000, E1   +47.497, E3 +313214.899}
SPL {X  -159.990, Y  +452.841, Z    +0.000, E1   +48.572, E3 +313227.746}
SPL {X  -159.990, Y  +439.038, Z    +0.000, E1   +49.804, E3 +313245.798}
SPL {X  -159.990, Y  +429.517, Z    +0.000, E1   +50.043, E3 +313261.146}
SPL {X  -159.990, Y  +423.834, Z    +0.000, E1   +50.037, E3 +313271.258}
SPL {X  -159.990, Y  +417.693, Z    +0.000, E1   +50.049, E3 +313282.156}
SPL {X  -159.990, Y  +411.447, Z    +0.000, E1   +50.039, E3 +313293.275}
SPL {X  -159.990, Y  +406.170, Z    +0.000, E1   +50.036, E3 +313302.647}
SPL {X  -159.990, Y  +399.787, Z    +0.000, E1   +50.064, E3 +313313.955}
SPL {X  -159.990, Y  +393.038, Z    +0.000, E1   +50.038, E3 +313325.989}
SPL {X  -159.990, Y  +387.356, Z    +0.000, E1   +50.042, E3 +313336.100}
SPL {X  -159.990, Y  +382.225, Z    +0.000, E1   +50.028, E3 +313345.245}
SPL {X  -159.846, Y  +375.718, Z    +0.000, E1   +50.041, E3 +313356.901}
SPL {X  -159.443, Y  +369.277, Z    +0.000, E1   +49.941, E3 +313368.815}
SPL {X  -158.871, Y  +363.614, Z    +0.000, E1   +49.855, E3 +313379.459}
SPL {X  -158.179, Y  +358.495, Z    +0.000, E1   +49.715, E3 +313389.308}
SPL {X  -157.077, Y  +352.107, Z    +0.000, E1   +49.567, E3 +313401.742}
SPL {X  -155.744, Y  +345.884, Z    +0.000, E1   +49.283, E3 +313414.229}
SPL {X  -154.686, Y  +341.646, Z    +0.000, E1   +49.094, E3 +313422.855}
SPL {X  -153.439, Y  +337.188, Z    +0.000, E1   +48.857, E3 +313432.062}
SPL {X  -151.836, Y  +332.074, Z    +0.000, E1   +48.585, E3 +313442.738}
SPL {X  -150.221, Y  +327.451, Z    +0.000, E1   +48.251, E3 +313452.616}
SPL {X  -148.587, Y  +323.181, Z    +0.000, E1   +47.960, E3 +313461.800}
SPL {X  -146.510, Y  +318.222, Z    +0.000, E1   +47.558, E3 +313472.636}
SPL {X  -141.189, Y  +307.250, Z    +0.000, E1   +40.067, E3 +313558.810}
ENDSPLINE

SPLINE
SPL {X  -154.923, Y  +342.556, Z    +0.000, E1   +23.930, E3 +313620.309}
SPL {X  -158.138, Y  +358.230, Z    +0.000, E1   +16.243, E3 +313629.267}
SPL {X  -159.647, Y  +372.034, Z    +0.000, E1    +8.739, E3 +313633.631}
SPL {X  -159.989, Y  +381.927, Z    +0.000, E1    +2.565, E3 +313635.391}
SPL {X  -159.990, Y  +386.909, Z    +0.000, E1    -1.211, E3 +313635.934}
SPL {X  -159.990, Y  +390.921, Z    +0.000, E1    -5.111, E3 +313636.413}
SPL {X  -159.990, Y  +395.719, Z    +0.000, E1   -10.396, E3 +313637.232}
SPL {X  -159.990, Y  +400.739, Z    +0.000, E1   -16.236, E3 +313638.430}
SPL {X  -159.990, Y  +409.482, Z    +0.000, E1   -25.418, E3 +313641.635}
SPL {X  -159.990, Y  +440.741, Z    +0.000, E1   -43.570, E3 +313662.292}
SPL {X  -159.990, Y  +489.732, Z    +0.000, E1   -48.863, E3 +313726.450}
SPL {X  -159.990, Y  +496.901, Z    +0.000, E1   -48.832, E3 +313739.797}
SPL {X  -159.990, Y  +502.531, Z    +0.000, E1   -48.834, E3 +313750.242}
SPL {X  -159.990, Y  +508.013, Z    +0.000, E1   -48.835, E3 +313760.377}
SPL {X  -159.990, Y  +513.813, Z    +0.000, E1   -48.843, E3 +313771.125}
SPL {X  -159.990, Y  +522.177, Z    +0.000, E1   -48.881, E3 +313786.602}
SPL {X  -159.990, Y  +532.076, Z    +0.000, E1   -48.872, E3 +313804.975}
SPL {X  -159.990, Y  +539.248, Z    +0.000, E1   -48.832, E3 +313818.343}
SPL {X  -159.990, Y  +544.926, Z    +0.000, E1   -48.835, E3 +313828.872}
SPL {X  -159.990, Y  +550.252, Z    +0.000, E1   -48.827, E3 +313838.778}
SPL {X  -159.990, Y  +555.692, Z    +0.000, E1   -48.830, E3 +313848.875}
SPL {X  -159.990, Y  +561.308, Z    +0.000, E1   -48.827, E3 +313859.322}
SPL {X  -159.990, Y  +566.669, Z    +0.000, E1   -48.820, E3 +313869.271}
SPL {X  -159.990, Y  +572.248, Z    +0.000, E1   -48.830, E3 +313879.616}
SPL {X  -159.990, Y  +577.770, Z    +0.000, E1   -48.821, E3 +313889.863}
SPL {X  -159.990, Y  +583.108, Z    +0.000, E1   -48.828, E3 +313899.765}
SPL {X  -159.990, Y  +588.804, Z    +0.000, E1   -48.829, E3 +313910.322}
SPL {X  -159.990, Y  +594.280, Z    +0.000, E1   -48.826, E3 +313920.484}
SPL {X  -159.990, Y  +600.107, Z    +0.000, E1   -48.833, E3 +313931.298}
SPL {X  -159.990, Y  +605.910, Z    +0.000, E1   -48.823, E3 +313942.077}
SPL {X  -159.990, Y  +611.566, Z    +0.000, E1   -48.829, E3 +313952.566}
SPL {X  -159.990, Y  +617.357, Z    +0.000, E1   -48.824, E3 +313963.321}
SPL {X  -159.990, Y  +622.965, Z    +0.000, E1   -48.826, E3 +313973.720}
SPL {X  -159.990, Y  +629.255, Z    +0.000, E1   -48.834, E3 +313985.387}
SPL {X  -159.990, Y  +634.905, Z    +0.000, E1   -48.821, E3 +313995.884}
SPL {X  -159.990, Y  +640.372, Z    +0.000, E1   -48.828, E3 +314006.021}
SPL {X  -159.990, Y  +646.939, Z    +0.000, E1   -48.838, E3 +314018.191}
SPL {X  -159.990, Y  +653.448, Z    +0.000, E1   -48.827, E3 +314030.286}
SPL {X  -159.990, Y  +659.039, Z    +0.000, E1   -48.826, E3 +314040.650}
SPL {X  -159.990, Y  +664.817, Z    +0.000, E1   -48.832, E3 +314051.365}
SPL {X  -159.990, Y  +671.221, Z    +0.000, E1   -48.836, E3 +314063.238}
SPL {X  -159.887, Y  +677.230, Z    +0.000, E1   -48.811, E3 +314074.504}
SPL {X  -159.602, Y  +682.629, Z    +0.000, E1   -48.761, E3 +314084.837}
SPL {X  -159.150, Y  +687.876, Z    +0.000, E1   -48.673, E3 +314095.076}
SPL {X  -158.569, Y  +692.776, Z    +0.000, E1   -48.570, E3 +314104.784}
SPL {X  -157.870, Y  +697.458, Z    +0.000, E1   -48.439, E3 +314114.213}
SPL {X  -157.028, Y  +702.144, Z    +0.000, E1   -48.297, E3 +314123.761}
SPL {X  -155.977, Y  +707.110, Z    +0.000, E1   -48.106, E3 +314134.065}
SPL {X  -154.657, Y  +712.464, Z    +0.000, E1   -47.874, E3 +314145.349}
SPL {X  -153.406, Y  +716.924, Z    +0.000, E1   -47.628, E3 +314154.915}
SPL {X  -152.020, Y  +721.367, Z    +0.000, E1   -47.374, E3 +314164.566}
SPL {X  -150.440, Y  +725.947, Z    +0.000, E1   -47.070, E3 +314174.671}
SPL {X  -148.730, Y  +730.459, Z    +0.000, E1   -46.749, E3 +314184.722}
SPL {X  -147.178, Y  +734.233, Z    +0.000, E1   -46.439, E3 +314193.256}
SPL {X  -140.263, Y  +748.461, Z    +0.000, E1   -42.675, E3 +314251.594}
ENDSPLINE

SPLINE
SPL {X  -141.835, Y  +745.525, Z    +0.000, E1   -39.068, E3 +314283.595}
SPL {X  -152.406, Y  +720.176, Z    +0.000, E1   -27.814, E3 +314334.808}
SPL {X  -157.542, Y  +699.382, Z    +0.000, E1   -18.086, E3 +314349.141}
SPL {X  -159.386, Y  +685.393, Z    +0.000, E1   -10.664, E3 +314354.095}
SPL {X  -159.928, Y  +675.946, Z    +0.000, E1    -5.007, E3 +314356.134}
SPL {X  -159.990, Y  +671.468, Z    +0.000, E1    -2.030, E3 +314356.730}
SPL {X  -159.990, Y  +667.678, Z    +0.000, E1    +0.783, E3 +314357.080}
SPL {X  -159.990, Y  +663.139, Z    +0.000, E1    +5.135, E3 +314357.597}
SPL {X  -159.990, Y  +658.551, Z    +0.000, E1   +10.313, E3 +314358.371}
SPL {X  -159.990, Y  +653.526, Z    +0.000, E1   +16.156, E3 +314359.606}
SPL {X  -159.990, Y  +644.434, Z    +0.000, E1   +25.921, E3 +314362.801}
SPL {X  -159.990, Y  +612.255, Z    +0.000, E1   +44.102, E3 +314384.682}
SPL {X  -159.990, Y  +561.053, Z    +0.000, E1   +49.668, E3 +314449.515}
SPL {X  -159.990, Y  +552.984, Z    +0.000, E1   +49.619, E3 +314464.156}
SPL {X  -159.990, Y  +547.278, Z    +0.000, E1   +49.619, E3 +314474.455}
SPL {X  -159.990, Y  +538.738, Z    +0.000, E1   +49.672, E3 +314489.779}
SPL {X  -159.990, Y  +529.436, Z    +0.000, E1   +49.638, E3 +314506.603}
SPL {X  -159.990, Y  +520.280, Z    +0.000, E1   +49.665, E3 +314523.082}
SPL {X  -159.990, Y  +511.038, Z    +0.000, E1   +49.636, E3 +314539.832}
SPL {X  -159.990, Y  +504.260, Z    +0.000, E1   +49.614, E3 +314552.105}
SPL {X  -159.990, Y  +503.881, Z    +0.000, E1   +48.376, E3 +314560.092}
ENDSPLINE

SPLINE
SPL {X  -159.990, Y  +520.622, Z    +0.000, E1   +41.395, E3 +314566.672}
ENDSPLINE

SPLINE
SPL {X  -159.990, Y  +512.735, Z    +0.000, E1   +42.369, E3 +314579.523}
SPL {X  -159.990, Y  +505.924, Z    +0.000, E1   +43.199, E3 +314590.181}
SPL {X  -159.990, Y  +497.983, Z    +0.000, E1   +44.027, E3 +314603.054}
SPL {X  -159.990, Y  +489.703, Z    +0.000, E1   +44.938, E3 +314615.473}
SPL {X  -159.990, Y  +484.712, Z    +0.000, E1   +45.426, E3 +314623.087}
SPL {X  -159.990, Y  +477.648, Z    +0.000, E1   +46.080, E3 +314633.907}
SPL {X  -159.990, Y  +469.952, Z    +0.000, E1   +46.750, E3 +314645.415}
SPL {X  -159.990, Y  +462.892, Z    +0.000, E1   +47.497, E3 +314654.899}
SPL {X  -159.990, Y  +450.424, Z    +0.000, E1   +48.824, E3 +314670.863}
SPL {X  -159.990, Y  +436.919, Z    +0.000, E1   +49.944, E3 +314688.632}
SPL {X  -159.990, Y  +429.517, Z    +0.000, E1   +50.043, E3 +314701.146}
SPL {X  -159.990, Y  +423.834, Z    +0.000, E1   +50.037, E3 +314711.258}
SPL {X  -159.990, Y  +417.693, Z    +0.000, E1   +50.049, E3 +314722.156}
SPL {X  -159.990, Y  +408.922, Z    +0.000, E1   +50.085, E3 +314737.686}
SPL {X  -159.990, Y  +399.787, Z    +0.000, E1   +50.064, E3 +314753.955}
SPL {X  -159.990, Y  +393.038, Z    +0.000, E1   +50.038, E3 +314765.989}
SPL {X  -159.990, Y  +385.182, Z    +0.000, E1   +50.081, E3 +314779.906}
SPL {X  -159.906, Y  +377.302, Z    +0.000, E1   +50.024, E3 +314794.067}
SPL {X  -159.545, Y  +370.569, Z    +0.000, E1   +49.982, E3 +314806.380}
SPL {X  -158.871, Y  +363.614, Z    +0.000, E1   +49.855, E3 +314819.459}
SPL {X  -158.179, Y  +358.495, Z    +0.000, E1   +49.715, E3 +314829.308}
SPL {X  -157.354, Y  +353.576, Z    +0.000, E1   +49.583, E3 +314838.894}
SPL {X  -156.029, Y  +347.121, Z    +0.000, E1   +49.358, E3 +314851.711}
SPL {X  -154.686, Y  +341.646, Z    +0.000, E1   +49.094, E3 +314862.855}
SPL {X  -153.089, Y  +336.017, Z    +0.000, E1   +48.817, E3 +314874.464}
SPL {X  -150.861, Y  +329.230, Z    +0.000, E1   +48.419, E3 +314888.753}
SPL {X  -148.587, Y  +323.181, Z    +0.000, E1   +47.960, E3 +314901.800}
SPL {X  -146.510, Y  +318.222, Z    +0.000, E1   +47.558, E3 +314912.636}
SPL {X  -141.189, Y  +307.250, Z    +0.000, E1   +40.067, E3 +314998.810}
ENDSPLINE

SPLINE
SPL {X  -154.923, Y  +342.556, Z    +0.000, E1   +23.930, E3 +315060.309}
SPL {X  -158.138, Y  +358.230, Z    +0.000, E1   +16.243, E3 +315069.267}
SPL {X  -159.407, Y  +368.849, Z    +0.000, E1   +10.504, E3 +315072.867}
SPL {X  -159.931, Y  +378.162, Z    +0.000, E1    +5.020, E3 +315074.852}
SPL {X  -159.990, Y  +384.616, Z    +0.000, E1    +0.627, E3 +315075.691}
SPL {X  -159.990, Y  +387.962, Z    +0.000, E1    -2.241, E3 +315076.048}
SPL {X  -159.990, Y  +390.921, Z    +0.000, E1    -5.111, E3 +315076.413}
SPL {X  -159.990, Y  +395.719, Z    +0.000, E1   -10.396, E3 +315077.232}
SPL {X  -159.990, Y  +400.739, Z    +0.000, E1   -16.236, E3 +315078.430}
SPL {X  -159.990, Y  +409.482, Z    +0.000, E1   -25.418, E3 +315081.635}
SPL {X  -159.990, Y  +440.741, Z    +0.000, E1   -43.570, E3 +315102.292}
SPL {X  -159.990, Y  +489.732, Z    +0.000, E1   -48.863, E3 +315166.450}
SPL {X  -159.990, Y  +496.901, Z    +0.000, E1   -48.832, E3 +315179.797}
SPL {X  -159.990, Y  +502.531, Z    +0.000, E1   -48.834, E3 +315190.242}
SPL {X  -159.990, Y  +508.013, Z    +0.000, E1   -48.835, E3 +315200.377}
SPL {X  -159.990, Y  +513.813, Z    +0.000, E1   -48.843, E3 +315211.125}
SPL {X  -159.990, Y  +522.177, Z    +0.000, E1   -48.881, E3 +315226.602}
SPL {X  -159.990, Y  +532.076, Z    +0.000, E1   -48.872, E3 +315244.975}
SPL {X  -159.990, Y  +539.248, Z    +0.000, E1   -48.832, E3 +315258.343}
SPL {X  -159.990, Y  +544.926, Z    +0.000, E1   -48.835, E3 +315268.872}
SPL {X  -159.990, Y  +550.252, Z    +0.000, E1   -48.827, E3 +315278.778}
SPL {X  -159.990, Y  +555.692, Z    +0.000, E1   -48.830, E3 +315288.875}
SPL {X  -159.990, Y  +561.308, Z    +0.000, E1   -48.827, E3 +315299.322}
SPL {X  -159.990, Y  +566.669, Z    +0.000, E1   -48.820, E3 +315309.271}
SPL {X  -159.990, Y  +572.248, Z    +0.000, E1   -48.830, E3 +315319.616}
SPL {X  -159.990, Y  +577.770, Z    +0.000, E1   -48.821, E3 +315329.863}
SPL {X  -159.990, Y  +583.108, Z    +0.000, E1   -48.828, E3 +315339.765}
SPL {X  -159.990, Y  +588.804, Z    +0.000, E1   -48.829, E3 +315350.322}
SPL {X  -159.990, Y  +594.280, Z    +0.000, E1   -48.826, E3 +315360.484}
SPL {X  -159.990, Y  +600.107, Z    +0.000, E1   -48.833, E3 +315371.298}
SPL {X  -159.990, Y  +605.910, Z    +0.000, E1   -48.823, E3 +315382.077}
SPL {X  -159.990, Y  +611.566, Z    +0.000, E1   -48.829, E3 +315392.566}
SPL {X  -159.990, Y  +617.357, Z    +0.000, E1   -48.824, E3 +315403.321}
SPL {X  -159.990, Y  +622.965, Z    +0.000, E1   -48.826, E3 +315413.720}
SPL {X  -159.990, Y  +629.255, Z    +0.000, E1   -48.834, E3 +315425.387}
SPL {X  -159.990, Y  +634.905, Z    +0.000, E1   -48.821, E3 +315435.884}
SPL {X  -159.990, Y  +640.372, Z    +0.000, E1   -48.828, E3 +315446.021}
SPL {X  -159.990, Y  +646.939, Z    +0.000, E1   -48.838, E3 +315458.191}
SPL {X  -159.990, Y  +653.448, Z    +0.000, E1   -48.827, E3 +315470.286}
SPL {X  -159.990, Y  +659.039, Z    +0.000, E1   -48.826, E3 +315480.650}
SPL {X  -159.990, Y  +664.817, Z    +0.000, E1   -48.832, E3 +315491.365}
SPL {X  -159.990, Y  +671.221, Z    +0.000, E1   -48.836, E3 +315503.238}
SPL {X  -159.887, Y  +677.230, Z    +0.000, E1   -48.811, E3 +315514.504}
SPL {X  -159.602, Y  +682.629, Z    +0.000, E1   -48.761, E3 +315524.837}
SPL {X  -159.150, Y  +687.876, Z    +0.000, E1   -48.673, E3 +315535.076}
SPL {X  -158.569, Y  +692.776, Z    +0.000, E1   -48.570, E3 +315544.784}
SPL {X  -157.870, Y  +697.458, Z    +0.000, E1   -48.439, E3 +315554.213}
SPL {X  -157.028, Y  +702.144, Z    +0.000, E1   -48.297, E3 +315563.761}
SPL {X  -155.977, Y  +707.110, Z    +0.000, E1   -48.106, E3 +315574.065}
SPL {X  -154.657, Y  +712.464, Z    +0.000, E1   -47.874, E3 +315585.349}
SPL {X  -153.406, Y  +716.924, Z    +0.000, E1   -47.628, E3 +315594.915}
SPL {X  -152.020, Y  +721.367, Z    +0.000, E1   -47.374, E3 +315604.566}
SPL {X  -150.440, Y  +725.947, Z    +0.000, E1   -47.070, E3 +315614.671}
SPL {X  -148.730, Y  +730.459, Z    +0.000, E1   -46.749, E3 +315624.722}
SPL {X  -147.178, Y  +734.233, Z    +0.000, E1   -46.439, E3 +315633.256}
SPL {X  -140.263, Y  +748.461, Z    +0.000, E1   -42.675, E3 +315691.594}
ENDSPLINE

SPLINE
SPL {X  -141.835, Y  +745.525, Z    +0.000, E1   -39.068, E3 +315723.595}
SPL {X  -152.406, Y  +720.176, Z    +0.000, E1   -27.814, E3 +315774.808}
SPL {X  -157.542, Y  +699.382, Z    +0.000, E1   -18.086, E3 +315789.141}
SPL {X  -159.386, Y  +685.393, Z    +0.000, E1   -10.664, E3 +315794.095}
SPL {X  -159.928, Y  +675.946, Z    +0.000, E1    -5.007, E3 +315796.134}
SPL {X  -159.990, Y  +671.468, Z    +0.000, E1    -2.030, E3 +315796.730}
SPL {X  -159.990, Y  +667.678, Z    +0.000, E1    +0.783, E3 +315797.080}
SPL {X  -159.990, Y  +663.139, Z    +0.000, E1    +5.135, E3 +315797.597}
SPL {X  -159.990, Y  +658.551, Z    +0.000, E1   +10.313, E3 +315798.371}
SPL {X  -159.990, Y  +653.526, Z    +0.000, E1   +16.156, E3 +315799.606}
SPL {X  -159.990, Y  +644.434, Z    +0.000, E1   +25.921, E3 +315802.801}
SPL {X  -159.990, Y  +612.255, Z    +0.000, E1   +44.102, E3 +315824.682}
SPL {X  -159.990, Y  +561.053, Z    +0.000, E1   +49.668, E3 +315889.515}
SPL {X  -159.990, Y  +552.984, Z    +0.000, E1   +49.619, E3 +315904.156}
SPL {X  -159.990, Y  +547.278, Z    +0.000, E1   +49.619, E3 +315914.455}
SPL {X  -159.990, Y  +538.738, Z    +0.000, E1   +49.672, E3 +315929.779}
SPL {X  -159.990, Y  +529.436, Z    +0.000, E1   +49.638, E3 +315946.603}
SPL {X  -159.990, Y  +520.280, Z    +0.000, E1   +49.665, E3 +315963.082}
SPL {X  -159.990, Y  +511.038, Z    +0.000, E1   +49.636, E3 +315979.832}
SPL {X  -159.990, Y  +504.260, Z    +0.000, E1   +49.614, E3 +315992.105}
SPL {X  -159.990, Y  +503.881, Z    +0.000, E1   +48.376, E3 +316000.092}
ENDSPLINE

SPLINE
SPL {X  -159.990, Y  +520.622, Z    +0.000, E1   +41.395, E3 +316006.672}
ENDSPLINE

SPLINE
SPL {X  -159.990, Y  +512.735, Z    +0.000, E1   +42.369, E3 +316019.523}
SPL {X  -159.990, Y  +505.924, Z    +0.000, E1   +43.199, E3 +316030.181}
SPL {X  -159.990, Y  +497.983, Z    +0.000, E1   +44.027, E3 +316043.054}
SPL {X  -159.990, Y  +489.703, Z    +0.000, E1   +44.938, E3 +316055.473}
SPL {X  -159.990, Y  +484.712, Z    +0.000, E1   +45.426, E3 +316063.087}
SPL {X  -159.990, Y  +477.648, Z    +0.000, E1   +46.080, E3 +316073.907}
SPL {X  -159.990, Y  +469.952, Z    +0.000, E1   +46.750, E3 +316085.415}
SPL {X  -159.990, Y  +462.892, Z    +0.000, E1   +47.497, E3 +316094.899}
SPL {X  -159.990, Y  +450.424, Z    +0.000, E1   +48.824, E3 +316110.863}
SPL {X  -159.990, Y  +436.919, Z    +0.000, E1   +49.944, E3 +316128.632}
SPL {X  -159.990, Y  +429.517, Z    +0.000, E1   +50.043, E3 +316141.146}
SPL {X  -159.990, Y  +423.834, Z    +0.000, E1   +50.037, E3 +316151.258}
SPL {X  -159.990, Y  +417.693, Z    +0.000, E1   +50.049, E3 +316162.156}
SPL {X  -159.990, Y  +408.922, Z    +0.000, E1   +50.085, E3 +316177.686}
SPL {X  -159.990, Y  +399.787, Z    +0.000, E1   +50.064, E3 +316193.955}
SPL {X  -159.990, Y  +393.038, Z    +0.000, E1   +50.038, E3 +316205.989}
SPL {X  -159.990, Y  +385.182, Z    +0.000, E1   +50.081, E3 +316219.906}
SPL {X  -159.906, Y  +377.302, Z    +0.000, E1   +50.024, E3 +316234.067}
SPL {X  -159.545, Y  +370.569, Z    +0.000, E1   +49.982, E3 +316246.380}
SPL {X  -158.871, Y  +363.614, Z    +0.000, E1   +49.855, E3 +316259.459}
SPL {X  -158.179, Y  +358.495, Z    +0.000, E1   +49.715, E3 +316269.308}
SPL {X  -157.354, Y  +353.576, Z    +0.000, E1   +49.583, E3 +316278.894}
SPL {X  -156.029, Y  +347.121, Z    +0.000, E1   +49.358, E3 +316291.711}
SPL {X  -154.686, Y  +341.646, Z    +0.000, E1   +49.094, E3 +316302.855}
SPL {X  -153.089, Y  +336.017, Z    +0.000, E1   +48.817, E3 +316314.464}
SPL {X  -151.481, Y  +331.019, Z    +0.000, E1   +48.491, E3 +316325.012}
SPL {X  -149.787, Y  +326.281, Z    +0.000, E1   +48.192, E3 +316335.100}
SPL {X  -148.124, Y  +322.035, Z    +0.000, E1   +47.846, E3 +316344.324}
SPL {X  -146.510, Y  +318.222, Z    +0.000, E1   +47.558, E3 +316352.636}
SPL {X  -141.189, Y  +307.250, Z    +0.000, E1   +40.067, E3 +316438.810}
ENDSPLINE

SPLINE
SPL {X  -154.923, Y  +342.556, Z    +0.000, E1   +23.930, E3 +316500.309}
SPL {X  -158.138, Y  +358.230, Z    +0.000, E1   +16.243, E3 +316509.267}
SPL {X  -159.647, Y  +372.034, Z    +0.000, E1    +8.739, E3 +316513.631}
SPL {X  -159.989, Y  +381.927, Z    +0.000, E1    +2.565, E3 +316515.391}
SPL {X  -159.990, Y  +386.909, Z    +0.000, E1    -1.211, E3 +316515.934}
SPL {X  -159.990, Y  +390.921, Z    +0.000, E1    -5.111, E3 +316516.413}
SPL {X  -159.990, Y  +395.719, Z    +0.000, E1   -10.396, E3 +316517.232}
SPL {X  -159.990, Y  +400.739, Z    +0.000, E1   -16.236, E3 +316518.430}
SPL {X  -159.990, Y  +409.482, Z    +0.000, E1   -25.418, E3 +316521.635}
SPL {X  -159.990, Y  +440.741, Z    +0.000, E1   -43.570, E3 +316542.292}
SPL {X  -159.990, Y  +489.732, Z    +0.000, E1   -48.863, E3 +316606.450}
SPL {X  -159.990, Y  +496.901, Z    +0.000, E1   -48.832, E3 +316619.797}
SPL {X  -159.990, Y  +502.531, Z    +0.000, E1   -48.834, E3 +316630.242}
SPL {X  -159.990, Y  +508.013, Z    +0.000, E1   -48.835, E3 +316640.377}
SPL {X  -159.990, Y  +513.813, Z    +0.000, E1   -48.843, E3 +316651.125}
SPL {X  -159.990, Y  +522.177, Z    +0.000, E1   -48.881, E3 +316666.602}
SPL {X  -159.990, Y  +532.076, Z    +0.000, E1   -48.872, E3 +316684.975}
SPL {X  -159.990, Y  +539.248, Z    +0.000, E1   -48.832, E3 +316698.343}
SPL {X  -159.990, Y  +544.926, Z    +0.000, E1   -48.835, E3 +316708.872}
SPL {X  -159.990, Y  +550.252, Z    +0.000, E1   -48.827, E3 +316718.778}
SPL {X  -159.990, Y  +555.692, Z    +0.000, E1   -48.830, E3 +316728.875}
SPL {X  -159.990, Y  +561.308, Z    +0.000, E1   -48.827, E3 +316739.322}
SPL {X  -159.990, Y  +566.669, Z    +0.000, E1   -48.820, E3 +316749.271}
SPL {X  -159.990, Y  +572.248, Z    +0.000, E1   -48.830, E3 +316759.616}
SPL {X  -159.990, Y  +577.770, Z    +0.000, E1   -48.821, E3 +316769.863}
SPL {X  -159.990, Y  +583.108, Z    +0.000, E1   -48.828, E3 +316779.765}
SPL {X  -159.990, Y  +588.804, Z    +0.000, E1   -48.829, E3 +316790.322}
SPL {X  -159.990, Y  +594.280, Z    +0.000, E1   -48.826, E3 +316800.484}
SPL {X  -159.990, Y  +600.107, Z    +0.000, E1   -48.833, E3 +316811.298}
SPL {X  -159.990, Y  +605.910, Z    +0.000, E1   -48.823, E3 +316822.077}
SPL {X  -159.990, Y  +611.566, Z    +0.000, E1   -48.829, E3 +316832.566}
SPL {X  -159.990, Y  +617.357, Z    +0.000, E1   -48.824, E3 +316843.321}
SPL {X  -159.990, Y  +622.965, Z    +0.000, E1   -48.826, E3 +316853.720}
SPL {X  -159.990, Y  +629.255, Z    +0.000, E1   -48.834, E3 +316865.387}
SPL {X  -159.990, Y  +634.905, Z    +0.000, E1   -48.821, E3 +316875.884}
SPL {X  -159.990, Y  +640.372, Z    +0.000, E1   -48.828, E3 +316886.021}
SPL {X  -159.990, Y  +646.939, Z    +0.000, E1   -48.838, E3 +316898.191}
SPL {X  -159.990, Y  +653.448, Z    +0.000, E1   -48.827, E3 +316910.286}
SPL {X  -159.990, Y  +659.039, Z    +0.000, E1   -48.826, E3 +316920.650}
SPL {X  -159.990, Y  +664.817, Z    +0.000, E1   -48.832, E3 +316931.365}
SPL {X  -159.990, Y  +671.221, Z    +0.000, E1   -48.836, E3 +316943.238}
SPL {X  -159.887, Y  +677.230, Z    +0.000, E1   -48.811, E3 +316954.504}
SPL {X  -159.602, Y  +682.629, Z    +0.000, E1   -48.761, E3 +316964.837}
SPL {X  -159.150, Y  +687.876, Z    +0.000, E1   -48.673, E3 +316975.076}
SPL {X  -158.569, Y  +692.776, Z    +0.000, E1   -48.570, E3 +316984.784}
SPL {X  -157.870, Y  +697.458, Z    +0.000, E1   -48.439, E3 +316994.213}
SPL {X  -157.028, Y  +702.144, Z    +0.000, E1   -48.297, E3 +317003.761}
SPL {X  -155.977, Y  +707.110, Z    +0.000, E1   -48.106, E3 +317014.065}
SPL {X  -154.657, Y  +712.464, Z    +0.000, E1   -47.874, E3 +317025.349}
SPL {X  -153.406, Y  +716.924, Z    +0.000, E1   -47.628, E3 +317034.915}
SPL {X  -152.020, Y  +721.367, Z    +0.000, E1   -47.374, E3 +317044.566}
SPL {X  -150.440, Y  +725.947, Z    +0.000, E1   -47.070, E3 +317054.671}
SPL {X  -148.730, Y  +730.459, Z    +0.000, E1   -46.749, E3 +317064.722}
SPL {X  -147.178, Y  +734.233, Z    +0.000, E1   -46.439, E3 +317073.256}
SPL {X  -140.222, Y  +748.536, Z    +0.000, E1   -42.074, E3 +317138.232}
ENDSPLINE

SPLINE
SPL {X  -152.021, Y  +721.365, Z    +0.000, E1   -28.339, E3 +317213.623}
SPL {X  -157.542, Y  +699.382, Z    +0.000, E1   -18.086, E3 +317229.141}
SPL {X  -159.386, Y  +685.393, Z    +0.000, E1   -10.664, E3 +317234.095}
SPL {X  -159.928, Y  +675.946, Z    +0.000, E1    -5.007, E3 +317236.134}
SPL {X  -159.990, Y  +671.468, Z    +0.000, E1    -2.030, E3 +317236.730}
SPL {X  -159.990, Y  +667.678, Z    +0.000, E1    +0.783, E3 +317237.080}
SPL {X  -159.990, Y  +663.139, Z    +0.000, E1    +5.135, E3 +317237.597}
SPL {X  -159.990, Y  +658.551, Z    +0.000, E1   +10.313, E3 +317238.371}
SPL {X  -159.990, Y  +653.526, Z    +0.000, E1   +16.156, E3 +317239.606}
SPL {X  -159.990, Y  +644.434, Z    +0.000, E1   +25.921, E3 +317242.801}
SPL {X  -159.990, Y  +612.255, Z    +0.000, E1   +44.102, E3 +317264.682}
SPL {X  -159.990, Y  +562.879, Z    +0.000, E1   +49.634, E3 +317326.271}
SPL {X  -159.990, Y  +554.544, Z    +0.000, E1   +49.649, E3 +317341.296}
SPL {X  -159.990, Y  +547.278, Z    +0.000, E1   +49.619, E3 +317354.455}
SPL {X  -159.990, Y  +540.489, Z    +0.000, E1   +49.634, E3 +317366.681}
SPL {X  -159.990, Y  +530.983, Z    +0.000, E1   +49.676, E3 +317383.752}
SPL {X  -159.990, Y  +522.804, Z    +0.000, E1   +49.620, E3 +317398.592}
SPL {X  -159.990, Y  +515.173, Z    +0.000, E1   +49.653, E3 +317412.330}
SPL {X  -159.990, Y  +505.472, Z    +0.000, E1   +49.465, E3 +317431.135}
ENDSPLINE

SPLINE
SPL {X  -159.990, Y  +518.841, Z    +0.000, E1   +41.643, E3 +317449.543}
ENDSPLINE

SPLINE
SPL {X  -159.990, Y  +508.096, Z    +0.000, E1   +42.952, E3 +317466.810}
SPL {X  -159.990, Y  +497.983, Z    +0.000, E1   +44.027, E3 +317483.054}
SPL {X  -159.990, Y  +489.703, Z    +0.000, E1   +44.938, E3 +317495.473}
SPL {X  -159.990, Y  +484.712, Z    +0.000, E1   +45.426, E3 +317503.087}
SPL {X  -159.990, Y  +477.648, Z    +0.000, E1   +46.080, E3 +317513.907}
SPL {X  -159.990, Y  +469.952, Z    +0.000, E1   +46.750, E3 +317525.415}
SPL {X  -159.990, Y  +460.762, Z    +0.000, E1   +47.755, E3 +317537.551}
SPL {X  -159.990, Y  +448.635, Z    +0.000, E1   +48.965, E3 +317553.239}
SPL {X  -159.990, Y  +436.919, Z    +0.000, E1   +49.944, E3 +317568.632}
SPL {X  -159.990, Y  +429.517, Z    +0.000, E1   +50.043, E3 +317581.146}
SPL {X  -159.990, Y  +421.718, Z    +0.000, E1   +50.072, E3 +317594.965}
SPL {X  -159.990, Y  +412.896, Z    +0.000, E1   +50.065, E3 +317610.658}
SPL {X  -159.990, Y  +406.170, Z    +0.000, E1   +50.036, E3 +317622.647}
SPL {X  -159.990, Y  +399.787, Z    +0.000, E1   +50.064, E3 +317633.955}
SPL {X  -159.990, Y  +393.038, Z    +0.000, E1   +50.038, E3 +317645.989}
SPL {X  -159.990, Y  +387.356, Z    +0.000, E1   +50.042, E3 +317656.100}
SPL {X  -159.956, Y  +379.183, Z    +0.000, E1   +50.071, E3 +317670.614}
SPL {X  -159.545, Y  +370.569, Z    +0.000, E1   +49.982, E3 +317686.380}
SPL {X  -158.871, Y  +363.614, Z    +0.000, E1   +49.855, E3 +317699.459}
SPL {X  -158.179, Y  +358.495, Z    +0.000, E1   +49.715, E3 +317709.308}
SPL {X  -157.077, Y  +352.107, Z    +0.000, E1   +49.567, E3 +317721.742}
SPL {X  -155.744, Y  +345.884, Z    +0.000, E1   +49.283, E3 +317734.229}
SPL {X  -154.686, Y  +341.646, Z    +0.000, E1   +49.094, E3 +317742.855}
SPL {X  -153.089, Y  +336.017, Z    +0.000, E1   +48.817, E3 +317754.464}
SPL {X  -151.481, Y  +331.019, Z    +0.000, E1   +48.491, E3 +317765.012}
SPL {X  -149.787, Y  +326.281, Z    +0.000, E1   +48.192, E3 +317775.100}
SPL {X  -148.124, Y  +322.035, Z    +0.000, E1   +47.846, E3 +317784.324}
SPL {X  -146.510, Y  +318.222, Z    +0.000, E1   +47.558, E3 +317792.636}
SPL {X  -141.189, Y  +307.250, Z    +0.000, E1   +40.067, E3 +317878.810}
ENDSPLINE

SPLINE
SPL {X  -154.923, Y  +342.556, Z    +0.000, E1   +23.930, E3 +317940.309}
SPL {X  -158.138, Y  +358.230, Z    +0.000, E1   +16.243, E3 +317949.267}
SPL {X  -159.647, Y  +372.034, Z    +0.000, E1    +8.739, E3 +317953.631}
SPL {X  -159.969, Y  +379.932, Z    +0.000, E1    +3.817, E3 +317955.139}
SPL {X  -159.990, Y  +384.616, Z    +0.000, E1    +0.627, E3 +317955.691}
SPL {X  -159.990, Y  +387.962, Z    +0.000, E1    -2.241, E3 +317956.048}
SPL {X  -159.990, Y  +390.921, Z    +0.000, E1    -5.111, E3 +317956.413}
SPL {X  -159.990, Y  +395.719, Z    +0.000, E1   -10.396, E3 +317957.232}
SPL {X  -159.990, Y  +400.739, Z    +0.000, E1   -16.236, E3 +317958.430}
SPL {X  -159.990, Y  +409.482, Z    +0.000, E1   -25.418, E3 +317961.635}
SPL {X  -159.990, Y  +440.741, Z    +0.000, E1   -43.570, E3 +317982.292}
SPL {X  -159.990, Y  +488.072, Z    +0.000, E1   -48.834, E3 +318043.414}
SPL {X  -159.990, Y  +495.397, Z    +0.000, E1   -48.860, E3 +318056.963}
SPL {X  -159.990, Y  +502.531, Z    +0.000, E1   -48.834, E3 +318070.242}
SPL {X  -159.990, Y  +508.013, Z    +0.000, E1   -48.835, E3 +318080.377}
SPL {X  -159.990, Y  +513.813, Z    +0.000, E1   -48.843, E3 +318091.125}
SPL {X  -159.990, Y  +522.177, Z    +0.000, E1   -48.881, E3 +318106.602}
SPL {X  -159.990, Y  +532.076, Z    +0.000, E1   -48.872, E3 +318124.975}
SPL {X  -159.990, Y  +539.248, Z    +0.000, E1   -48.832, E3 +318138.343}
SPL {X  -159.990, Y  +544.926, Z    +0.000, E1   -48.835, E3 +318148.872}
SPL {X  -159.990, Y  +550.252, Z    +0.000, E1   -48.827, E3 +318158.778}
SPL {X  -159.990, Y  +555.692, Z    +0.000, E1   -48.830, E3 +318168.875}
SPL {X  -159.990, Y  +561.308, Z    +0.000, E1   -48.827, E3 +318179.322}
SPL {X  -159.990, Y  +566.669, Z    +0.000, E1   -48.820, E3 +318189.271}
SPL {X  -159.990, Y  +572.248, Z    +0.000, E1   -48.830, E3 +318199.616}
SPL {X  -159.990, Y  +577.770, Z    +0.000, E1   -48.821, E3 +318209.863}
SPL {X  -159.990, Y  +583.108, Z    +0.000, E1   -48.828, E3 +318219.765}
SPL {X  -159.990, Y  +588.804, Z    +0.000, E1   -48.829, E3 +318230.322}
SPL {X  -159.990, Y  +594.280, Z    +0.000, E1   -48.826, E3 +318240.484}
SPL {X  -159.990, Y  +600.107, Z    +0.000, E1   -48.833, E3 +318251.298}
SPL {X  -159.990, Y  +605.910, Z    +0.000, E1   -48.823, E3 +318262.077}
SPL {X  -159.990, Y  +611.566, Z    +0.000, E1   -48.829, E3 +318272.566}
SPL {X  -159.990, Y  +617.357, Z    +0.000, E1   -48.824, E3 +318283.321}
SPL {X  -159.990, Y  +622.965, Z    +0.000, E1   -48.826, E3 +318293.720}
SPL {X  -159.990, Y  +629.255, Z    +0.000, E1   -48.834, E3 +318305.387}
SPL {X  -159.990, Y  +634.905, Z    +0.000, E1   -48.821, E3 +318315.884}
SPL {X  -159.990, Y  +640.372, Z    +0.000, E1   -48.828, E3 +318326.021}
SPL {X  -159.990, Y  +646.939, Z    +0.000, E1   -48.838, E3 +318338.191}
SPL {X  -159.990, Y  +653.448, Z    +0.000, E1   -48.827, E3 +318350.286}
SPL {X  -159.990, Y  +659.039, Z    +0.000, E1   -48.826, E3 +318360.650}
SPL {X  -159.990, Y  +664.817, Z    +0.000, E1   -48.832, E3 +318371.365}
SPL {X  -159.990, Y  +671.221, Z    +0.000, E1   -48.836, E3 +318383.238}
SPL {X  -159.887, Y  +677.230, Z    +0.000, E1   -48.811, E3 +318394.504}
SPL {X  -159.602, Y  +682.629, Z    +0.000, E1   -48.761, E3 +318404.837}
SPL {X  -159.150, Y  +687.876, Z    +0.000, E1   -48.673, E3 +318415.076}
SPL {X  -158.569, Y  +692.776, Z    +0.000, E1   -48.570, E3 +318424.784}
SPL {X  -157.870, Y  +697.458, Z    +0.000, E1   -48.439, E3 +318434.213}
SPL {X  -157.028, Y  +702.144, Z    +0.000, E1   -48.297, E3 +318443.761}
SPL {X  -155.977, Y  +707.110, Z    +0.000, E1   -48.106, E3 +318454.065}
SPL {X  -154.657, Y  +712.464, Z    +0.000, E1   -47.874, E3 +318465.349}
SPL {X  -153.406, Y  +716.924, Z    +0.000, E1   -47.628, E3 +318474.915}
SPL {X  -152.020, Y  +721.367, Z    +0.000, E1   -47.374, E3 +318484.566}
SPL {X  -150.440, Y  +725.947, Z    +0.000, E1   -47.070, E3 +318494.671}
SPL {X  -148.730, Y  +730.459, Z    +0.000, E1   -46.749, E3 +318504.722}
SPL {X  -147.178, Y  +734.233, Z    +0.000, E1   -46.439, E3 +318513.256}
SPL {X  -140.222, Y  +748.536, Z    +0.000, E1   -42.074, E3 +318578.232}
ENDSPLINE

SPLINE
SPL {X  -152.021, Y  +721.365, Z    +0.000, E1   -28.339, E3 +318653.623}
SPL {X  -158.165, Y  +695.595, Z    +0.000, E1   -16.189, E3 +318670.706}
SPL {X  -159.572, Y  +683.063, Z    +0.000, E1    -9.282, E3 +318674.713}
SPL {X  -159.928, Y  +675.946, Z    +0.000, E1    -5.007, E3 +318676.134}
SPL {X  -159.990, Y  +669.697, Z    +0.000, E1    -0.851, E3 +318676.894}
SPL {X  -159.990, Y  +665.698, Z    +0.000, E1    +2.616, E3 +318677.273}
SPL {X  -159.990, Y  +660.480, Z    +0.000, E1    +7.942, E3 +318678.031}
SPL {X  -159.990, Y  +653.526, Z    +0.000, E1   +16.156, E3 +318679.606}
SPL {X  -159.990, Y  +644.434, Z    +0.000, E1   +25.921, E3 +318682.801}
SPL {X  -159.990, Y  +612.255, Z    +0.000, E1   +44.102, E3 +318704.682}
SPL {X  -159.990, Y  +562.879, Z    +0.000, E1   +49.634, E3 +318766.271}
SPL {X  -159.990, Y  +554.544, Z    +0.000, E1   +49.649, E3 +318781.296}
SPL {X  -159.990, Y  +547.278, Z    +0.000, E1   +49.619, E3 +318794.455}
SPL {X  -159.990, Y  +540.489, Z    +0.000, E1   +49.634, E3 +318806.681}
SPL {X  -159.990, Y  +530.983, Z    +0.000, E1   +49.676, E3 +318823.752}
SPL {X  -159.990, Y  +522.804, Z    +0.000, E1   +49.620, E3 +318838.592}
SPL {X  -159.990, Y  +515.173, Z    +0.000, E1   +49.653, E3 +318852.330}
SPL {X  -159.990, Y  +505.472, Z    +0.000, E1   +49.465, E3 +318871.135}
ENDSPLINE

SPLINE
SPL {X  -159.990, Y  +518.841, Z    +0.000, E1   +41.643, E3 +318889.543}
ENDSPLINE

SPLINE
SPL {X  -159.990, Y  +508.096, Z    +0.000, E1   +42.952, E3 +318906.810}
SPL {X  -159.990, Y  +500.642, Z    +0.000, E1   +43.747, E3 +318918.731}
SPL {X  -159.990, Y  +495.820, Z    +0.000, E1   +44.207, E3 +318926.618}
SPL {X  -159.990, Y  +487.435, Z    +0.000, E1   +45.185, E3 +318938.910}
SPL {X  -159.990, Y  +477.648, Z    +0.000, E1   +46.080, E3 +318953.907}
SPL {X  -159.990, Y  +469.952, Z    +0.000, E1   +46.750, E3 +318965.415}
SPL {X  -159.990, Y  +460.762, Z    +0.000, E1   +47.755, E3 +318977.551}
SPL {X  -159.990, Y  +451.028, Z    +0.000, E1   +48.723, E3 +318990.163}
SPL {X  -159.990, Y  +441.023, Z    +0.000, E1   +49.655, E3 +319002.997}
SPL {X  -159.990, Y  +431.096, Z    +0.000, E1   +50.075, E3 +319018.285}
SPL {X  -159.990, Y  +423.834, Z    +0.000, E1   +50.037, E3 +319031.258}
SPL {X  -159.990, Y  +417.693, Z    +0.000, E1   +50.049, E3 +319042.156}
SPL {X  -159.990, Y  +411.447, Z    +0.000, E1   +50.039, E3 +319053.275}
SPL {X  -159.990, Y  +406.170, Z    +0.000, E1   +50.036, E3 +319062.647}
SPL {X  -159.990, Y  +399.787, Z    +0.000, E1   +50.064, E3 +319073.955}
SPL {X  -159.990, Y  +393.038, Z    +0.000, E1   +50.038, E3 +319085.989}
SPL {X  -159.990, Y  +387.356, Z    +0.000, E1   +50.042, E3 +319096.100}
SPL {X  -159.956, Y  +379.183, Z    +0.000, E1   +50.071, E3 +319110.614}
SPL {X  -159.413, Y  +368.921, Z    +0.000, E1   +49.998, E3 +319129.389}
SPL {X  -158.412, Y  +360.086, Z    +0.000, E1   +49.787, E3 +319146.191}
SPL {X  -157.077, Y  +352.107, Z    +0.000, E1   +49.567, E3 +319161.742}
SPL {X  -155.744, Y  +345.884, Z    +0.000, E1   +49.283, E3 +319174.229}
SPL {X  -154.686, Y  +341.646, Z    +0.000, E1   +49.094, E3 +319182.855}
SPL {X  -153.089, Y  +336.017, Z    +0.000, E1   +48.817, E3 +319194.464}
SPL {X  -151.481, Y  +331.019, Z    +0.000, E1   +48.491, E3 +319205.012}
SPL {X  -149.787, Y  +326.281, Z    +0.000, E1   +48.192, E3 +319215.100}
SPL {X  -148.124, Y  +322.035, Z    +0.000, E1   +47.846, E3 +319224.324}
SPL {X  -146.510, Y  +318.222, Z    +0.000, E1   +47.558, E3 +319232.636}
SPL {X  -141.189, Y  +307.250, Z    +0.000, E1   +40.067, E3 +319318.810}
ENDSPLINE

SPLINE
SPL {X  -154.923, Y  +342.556, Z    +0.000, E1   +23.930, E3 +319380.309}
SPL {X  -158.138, Y  +358.230, Z    +0.000, E1   +16.243, E3 +319389.267}
SPL {X  -159.407, Y  +368.849, Z    +0.000, E1   +10.504, E3 +319392.867}
SPL {X  -159.931, Y  +378.162, Z    +0.000, E1    +5.020, E3 +319394.852}
SPL {X  -159.990, Y  +384.616, Z    +0.000, E1    +0.627, E3 +319395.691}
SPL {X  -159.990, Y  +387.962, Z    +0.000, E1    -2.241, E3 +319396.048}
SPL {X  -159.990, Y  +390.921, Z    +0.000, E1    -5.111, E3 +319396.413}
SPL {X  -159.990, Y  +395.719, Z    +0.000, E1   -10.396, E3 +319397.232}
SPL {X  -159.990, Y  +400.739, Z    +0.000, E1   -16.236, E3 +319398.430}
SPL {X  -159.990, Y  +407.669, Z    +0.000, E1   -23.731, E3 +319400.753}
SPL {X  -159.990, Y  +417.102, Z    +0.000, E1   -32.094, E3 +319405.313}
SPL {X  -159.990, Y  +440.741, Z    +0.000, E1   -43.570, E3 +319422.292}
SPL {X  -159.990, Y  +488.072, Z    +0.000, E1   -48.834, E3 +319483.414}
SPL {X  -159.990, Y  +495.397, Z    +0.000, E1   -48.860, E3 +319496.963}
SPL {X  -159.990, Y  +502.531, Z    +0.000, E1   -48.834, E3 +319510.242}
SPL {X  -159.990, Y  +508.013, Z    +0.000, E1   -48.835, E3 +319520.377}
SPL {X  -159.990, Y  +513.813, Z    +0.000, E1   -48.843, E3 +319531.125}
SPL {X  -159.990, Y  +522.177, Z    +0.000, E1   -48.881, E3 +319546.602}
SPL {X  -159.990, Y  +532.076, Z    +0.000, E1   -48.872, E3 +319564.975}
SPL {X  -159.990, Y  +539.248, Z    +0.000, E1   -48.832, E3 +319578.343}
SPL {X  -159.990, Y  +544.926, Z    +0.000, E1   -48.835, E3 +319588.872}
SPL {X  -159.990, Y  +550.252, Z    +0.000, E1   -48.827, E3 +319598.778}
SPL {X  -159.990, Y  +555.692, Z    +0.000, E1   -48.830, E3 +319608.875}
SPL {X  -159.990, Y  +561.308, Z    +0.000, E1   -48.827, E3 +319619.322}
SPL {X  -159.990, Y  +566.669, Z    +0.000, E1   -48.820, E3 +319629.271}
SPL {X  -159.990, Y  +572.248, Z    +0.000, E1   -48.830, E3 +319639.616}
SPL {X  -159.990, Y  +577.770, Z    +0.000, E1   -48.821, E3 +319649.863}
SPL {X  -159.990, Y  +583.108, Z    +0.000, E1   -48.828, E3 +319659.765}
SPL {X  -159.990, Y  +588.804, Z    +0.000, E1   -48.829, E3 +319670.322}
SPL {X  -159.990, Y  +594.280, Z    +0.000, E1   -48.826, E3 +319680.484}
SPL {X  -159.990, Y  +600.107, Z    +0.000, E1   -48.833, E3 +319691.298}
SPL {X  -159.990, Y  +605.910, Z    +0.000, E1   -48.823, E3 +319702.077}
SPL {X  -159.990, Y  +611.566, Z    +0.000, E1   -48.829, E3 +319712.566}
SPL {X  -159.990, Y  +617.357, Z    +0.000, E1   -48.824, E3 +319723.321}
SPL {X  -159.990, Y  +622.965, Z    +0.000, E1   -48.826, E3 +319733.720}
SPL {X  -159.990, Y  +629.255, Z    +0.000, E1   -48.834, E3 +319745.387}
SPL {X  -159.990, Y  +634.905, Z    +0.000, E1   -48.821, E3 +319755.884}
SPL {X  -159.990, Y  +640.372, Z    +0.000, E1   -48.828, E3 +319766.021}
SPL {X  -159.990, Y  +646.939, Z    +0.000, E1   -48.838, E3 +319778.191}
SPL {X  -159.990, Y  +653.448, Z    +0.000, E1   -48.827, E3 +319790.286}
SPL {X  -159.990, Y  +659.039, Z    +0.000, E1   -48.826, E3 +319800.650}
SPL {X  -159.990, Y  +664.817, Z    +0.000, E1   -48.832, E3 +319811.365}
SPL {X  -159.990, Y  +671.221, Z    +0.000, E1   -48.836, E3 +319823.238}
SPL {X  -159.887, Y  +677.230, Z    +0.000, E1   -48.811, E3 +319834.504}
SPL {X  -159.602, Y  +682.629, Z    +0.000, E1   -48.761, E3 +319844.837}
SPL {X  -159.150, Y  +687.876, Z    +0.000, E1   -48.673, E3 +319855.076}
SPL {X  -158.569, Y  +692.776, Z    +0.000, E1   -48.570, E3 +319864.784}
SPL {X  -157.870, Y  +697.458, Z    +0.000, E1   -48.439, E3 +319874.213}
SPL {X  -157.028, Y  +702.144, Z    +0.000, E1   -48.297, E3 +319883.761}
SPL {X  -155.977, Y  +707.110, Z    +0.000, E1   -48.106, E3 +319894.065}
SPL {X  -154.657, Y  +712.464, Z    +0.000, E1   -47.874, E3 +319905.349}
SPL {X  -153.406, Y  +716.924, Z    +0.000, E1   -47.628, E3 +319914.915}
SPL {X  -152.020, Y  +721.367, Z    +0.000, E1   -47.374, E3 +319924.566}
SPL {X  -150.440, Y  +725.947, Z    +0.000, E1   -47.070, E3 +319934.671}
SPL {X  -148.730, Y  +730.459, Z    +0.000, E1   -46.749, E3 +319944.722}
SPL {X  -147.178, Y  +734.233, Z    +0.000, E1   -46.439, E3 +319953.256}
SPL {X  -140.263, Y  +748.461, Z    +0.000, E1   -42.675, E3 +320011.594}
ENDSPLINE

SPLINE
SPL {X  -141.835, Y  +745.525, Z    +0.000, E1   -39.068, E3 +320043.595}
SPL {X  -152.406, Y  +720.176, Z    +0.000, E1   -27.814, E3 +320094.808}
SPL {X  -158.165, Y  +695.595, Z    +0.000, E1   -16.189, E3 +320110.706}
SPL {X  -159.572, Y  +683.063, Z    +0.000, E1    -9.282, E3 +320114.713}
SPL {X  -159.928, Y  +675.946, Z    +0.000, E1    -5.007, E3 +320116.134}
SPL {X  -159.990, Y  +671.468, Z    +0.000, E1    -2.030, E3 +320116.730}
SPL {X  -159.990, Y  +667.678, Z    +0.000, E1    +0.783, E3 +320117.080}
SPL {X  -159.990, Y  +663.139, Z    +0.000, E1    +5.135, E3 +320117.597}
SPL {X  -159.990, Y  +658.551, Z    +0.000, E1   +10.313, E3 +320118.371}
SPL {X  -159.990, Y  +653.526, Z    +0.000, E1   +16.156, E3 +320119.606}
SPL {X  -159.990, Y  +644.434, Z    +0.000, E1   +25.921, E3 +320122.801}
SPL {X  -159.990, Y  +612.255, Z    +0.000, E1   +44.102, E3 +320144.682}
SPL {X  -159.990, Y  +562.879, Z    +0.000, E1   +49.634, E3 +320206.271}
SPL {X  -159.990, Y  +554.544, Z    +0.000, E1   +49.649, E3 +320221.296}
SPL {X  -159.990, Y  +547.278, Z    +0.000, E1   +49.619, E3 +320234.455}
SPL {X  -159.990, Y  +540.489, Z    +0.000, E1   +49.634, E3 +320246.681}
SPL {X  -159.990, Y  +532.689, Z    +0.000, E1   +49.639, E3 +320260.734}
SPL {X  -159.990, Y  +524.316, Z    +0.000, E1   +49.648, E3 +320275.819}
SPL {X  -159.990, Y  +515.173, Z    +0.000, E1   +49.653, E3 +320292.330}
SPL {X  -159.990, Y  +505.896, Z    +0.000, E1   +49.645, E3 +320309.105}
SPL {X  -159.990, Y  +503.881, Z    +0.000, E1   +48.376, E3 +320320.092}
ENDSPLINE

SPLINE
SPL {X  -159.990, Y  +520.622, Z    +0.000, E1   +41.395, E3 +320326.672}
ENDSPLINE

SPLINE
SPL {X  -159.990, Y  +512.735, Z    +0.000, E1   +42.369, E3 +320339.523}
SPL {X  -159.990, Y  +503.505, Z    +0.000, E1   +43.480, E3 +320354.068}
SPL {X  -159.990, Y  +492.511, Z    +0.000, E1   +44.632, E3 +320371.383}
SPL {X  -159.990, Y  +482.131, Z    +0.000, E1   +45.680, E3 +320387.053}
SPL {X  -159.990, Y  +472.111, Z    +0.000, E1   +46.581, E3 +320402.185}
SPL {X  -159.990, Y  +460.762, Z    +0.000, E1   +47.755, E3 +320417.551}
SPL {X  -159.990, Y  +448.635, Z    +0.000, E1   +48.965, E3 +320433.239}
SPL {X  -159.990, Y  +436.919, Z    +0.000, E1   +49.944, E3 +320448.632}
SPL {X  -159.990, Y  +429.517, Z    +0.000, E1   +50.043, E3 +320461.146}
SPL {X  -159.990, Y  +423.834, Z    +0.000, E1   +50.037, E3 +320471.258}
SPL {X  -159.990, Y  +417.693, Z    +0.000, E1   +50.049, E3 +320482.156}
SPL {X  -159.990, Y  +408.922, Z    +0.000, E1   +50.085, E3 +320497.686}
SPL {X  -159.990, Y  +399.787, Z    +0.000, E1   +50.064, E3 +320513.955}
SPL {X  -159.990, Y  +393.038, Z    +0.000, E1   +50.038, E3 +320525.989}
SPL {X  -159.990, Y  +385.182, Z    +0.000, E1   +50.081, E3 +320539.906}
SPL {X  -159.846, Y  +375.718, Z    +0.000, E1   +50.041, E3 +320556.901}
SPL {X  -159.300, Y  +367.653, Z    +0.000, E1   +49.944, E3 +320571.809}
SPL {X  -158.412, Y  +360.086, Z    +0.000, E1   +49.787, E3 +320586.191}
SPL {X  -157.077, Y  +352.107, Z    +0.000, E1   +49.567, E3 +320601.742}
SPL {X  -155.744, Y  +345.884, Z    +0.000, E1   +49.283, E3 +320614.229}
SPL {X  -154.686, Y  +341.646, Z    +0.000, E1   +49.094, E3 +320622.855}
SPL {X  -153.089, Y  +336.017, Z    +0.000, E1   +48.817, E3 +320634.464}
SPL {X  -150.861, Y  +329.230, Z    +0.000, E1   +48.419, E3 +320648.753}
SPL {X  -148.587, Y  +323.181, Z    +0.000, E1   +47.960, E3 +320661.800}
SPL {X  -146.510, Y  +318.222, Z    +0.000, E1   +47.558, E3 +320672.636}
SPL {X  -141.189, Y  +307.250, Z    +0.000, E1   +40.067, E3 +320758.810}
ENDSPLINE

SPLINE
SPL {X  -154.923, Y  +342.556, Z    +0.000, E1   +23.930, E3 +320820.309}
SPL {X  -158.138, Y  +358.230, Z    +0.000, E1   +16.243, E3 +320829.267}
SPL {X  -159.647, Y  +372.034, Z    +0.000, E1    +8.739, E3 +320833.631}
SPL {X  -159.989, Y  +381.927, Z    +0.000, E1    +2.565, E3 +320835.391}
SPL {X  -159.990, Y  +386.909, Z    +0.000, E1    -1.211, E3 +320835.934}
SPL {X  -159.990, Y  +390.921, Z    +0.000, E1    -5.111, E3 +320836.413}
SPL {X  -159.990, Y  +395.719, Z    +0.000, E1   -10.396, E3 +320837.232}
SPL {X  -159.990, Y  +400.739, Z    +0.000, E1   -16.236, E3 +320838.430}
SPL {X  -159.990, Y  +409.482, Z    +0.000, E1   -25.418, E3 +320841.635}
SPL {X  -159.990, Y  +440.741, Z    +0.000, E1   -43.570, E3 +320862.292}
SPL {X  -159.990, Y  +489.732, Z    +0.000, E1   -48.863, E3 +320926.450}
SPL {X  -159.990, Y  +496.901, Z    +0.000, E1   -48.832, E3 +320939.797}
SPL {X  -159.990, Y  +502.531, Z    +0.000, E1   -48.834, E3 +320950.242}
SPL {X  -159.990, Y  +508.013, Z    +0.000, E1   -48.835, E3 +320960.377}
SPL {X  -159.990, Y  +513.813, Z    +0.000, E1   -48.843, E3 +320971.125}
SPL {X  -159.990, Y  +522.177, Z    +0.000, E1   -48.881, E3 +320986.602}
SPL {X  -159.990, Y  +532.076, Z    +0.000, E1   -48.872, E3 +321004.975}
SPL {X  -159.990, Y  +539.248, Z    +0.000, E1   -48.832, E3 +321018.343}
SPL {X  -159.990, Y  +544.926, Z    +0.000, E1   -48.835, E3 +321028.872}
SPL {X  -159.990, Y  +550.252, Z    +0.000, E1   -48.827, E3 +321038.778}
SPL {X  -159.990, Y  +555.692, Z    +0.000, E1   -48.830, E3 +321048.875}
SPL {X  -159.990, Y  +561.308, Z    +0.000, E1   -48.827, E3 +321059.322}
SPL {X  -159.990, Y  +566.669, Z    +0.000, E1   -48.820, E3 +321069.271}
SPL {X  -159.990, Y  +572.248, Z    +0.000, E1   -48.830, E3 +321079.616}
SPL {X  -159.990, Y  +577.770, Z    +0.000, E1   -48.821, E3 +321089.863}
SPL {X  -159.990, Y  +583.108, Z    +0.000, E1   -48.828, E3 +321099.765}
SPL {X  -159.990, Y  +588.804, Z    +0.000, E1   -48.829, E3 +321110.322}
SPL {X  -159.990, Y  +594.280, Z    +0.000, E1   -48.826, E3 +321120.484}
SPL {X  -159.990, Y  +600.107, Z    +0.000, E1   -48.833, E3 +321131.298}
SPL {X  -159.990, Y  +605.910, Z    +0.000, E1   -48.823, E3 +321142.077}
SPL {X  -159.990, Y  +611.566, Z    +0.000, E1   -48.829, E3 +321152.566}
SPL {X  -159.990, Y  +617.357, Z    +0.000, E1   -48.824, E3 +321163.321}
SPL {X  -159.990, Y  +622.965, Z    +0.000, E1   -48.826, E3 +321173.720}
SPL {X  -159.990, Y  +629.255, Z    +0.000, E1   -48.834, E3 +321185.387}
SPL {X  -159.990, Y  +634.905, Z    +0.000, E1   -48.821, E3 +321195.884}
SPL {X  -159.990, Y  +640.372, Z    +0.000, E1   -48.828, E3 +321206.021}
SPL {X  -159.990, Y  +646.939, Z    +0.000, E1   -48.838, E3 +321218.191}
SPL {X  -159.990, Y  +653.448, Z    +0.000, E1   -48.827, E3 +321230.286}
SPL {X  -159.990, Y  +659.039, Z    +0.000, E1   -48.826, E3 +321240.650}
SPL {X  -159.990, Y  +664.817, Z    +0.000, E1   -48.832, E3 +321251.365}
SPL {X  -159.990, Y  +671.221, Z    +0.000, E1   -48.836, E3 +321263.238}
SPL {X  -159.887, Y  +677.230, Z    +0.000, E1   -48.811, E3 +321274.504}
SPL {X  -159.602, Y  +682.629, Z    +0.000, E1   -48.761, E3 +321284.837}
SPL {X  -159.150, Y  +687.876, Z    +0.000, E1   -48.673, E3 +321295.076}
SPL {X  -158.569, Y  +692.776, Z    +0.000, E1   -48.570, E3 +321304.784}
SPL {X  -157.870, Y  +697.458, Z    +0.000, E1   -48.439, E3 +321314.213}
SPL {X  -157.028, Y  +702.144, Z    +0.000, E1   -48.297, E3 +321323.761}
SPL {X  -155.977, Y  +707.110, Z    +0.000, E1   -48.106, E3 +321334.065}
SPL {X  -154.657, Y  +712.464, Z    +0.000, E1   -47.874, E3 +321345.349}
SPL {X  -153.406, Y  +716.924, Z    +0.000, E1   -47.628, E3 +321354.915}
SPL {X  -152.020, Y  +721.367, Z    +0.000, E1   -47.374, E3 +321364.566}
SPL {X  -150.440, Y  +725.947, Z    +0.000, E1   -47.070, E3 +321374.671}
SPL {X  -148.730, Y  +730.459, Z    +0.000, E1   -46.749, E3 +321384.722}
SPL {X  -147.178, Y  +734.233, Z    +0.000, E1   -46.439, E3 +321393.256}
SPL {X  -140.263, Y  +748.461, Z    +0.000, E1   -42.675, E3 +321451.594}
ENDSPLINE

SPLINE
SPL {X  -141.835, Y  +745.525, Z    +0.000, E1   -39.068, E3 +321483.595}
SPL {X  -152.406, Y  +720.176, Z    +0.000, E1   -27.814, E3 +321534.808}
SPL {X  -158.165, Y  +695.595, Z    +0.000, E1   -16.189, E3 +321550.706}
SPL {X  -159.572, Y  +683.063, Z    +0.000, E1    -9.282, E3 +321554.713}
SPL {X  -159.928, Y  +675.946, Z    +0.000, E1    -5.007, E3 +321556.134}
SPL {X  -159.990, Y  +669.697, Z    +0.000, E1    -0.851, E3 +321556.894}
SPL {X  -159.990, Y  +665.698, Z    +0.000, E1    +2.616, E3 +321557.273}
SPL {X  -159.990, Y  +662.251, Z    +0.000, E1    +6.155, E3 +321557.719}
SPL {X  -159.990, Y  +658.551, Z    +0.000, E1   +10.313, E3 +321558.371}
SPL {X  -159.990, Y  +653.526, Z    +0.000, E1   +16.156, E3 +321559.606}
SPL {X  -159.990, Y  +644.434, Z    +0.000, E1   +25.921, E3 +321562.801}
SPL {X  -159.990, Y  +612.255, Z    +0.000, E1   +44.102, E3 +321584.682}
SPL {X  -159.990, Y  +561.053, Z    +0.000, E1   +49.668, E3 +321649.515}
SPL {X  -159.990, Y  +552.984, Z    +0.000, E1   +49.619, E3 +321664.156}
SPL {X  -159.990, Y  +547.278, Z    +0.000, E1   +49.619, E3 +321674.455}
SPL {X  -159.990, Y  +538.738, Z    +0.000, E1   +49.672, E3 +321689.779}
SPL {X  -159.990, Y  +529.436, Z    +0.000, E1   +49.638, E3 +321706.603}
SPL {X  -159.990, Y  +522.804, Z    +0.000, E1   +49.620, E3 +321718.592}
SPL {X  -159.990, Y  +515.173, Z    +0.000, E1   +49.653, E3 +321732.330}
SPL {X  -159.990, Y  +505.472, Z    +0.000, E1   +49.465, E3 +321751.135}
ENDSPLINE

SPLINE
SPL {X  -159.990, Y  +518.841, Z    +0.000, E1   +41.643, E3 +321769.543}
ENDSPLINE

SPLINE
SPL {X  -159.990, Y  +508.096, Z    +0.000, E1   +42.952, E3 +321786.810}
SPL {X  -159.990, Y  +500.642, Z    +0.000, E1   +43.747, E3 +321798.731}
SPL {X  -159.990, Y  +495.820, Z    +0.000, E1   +44.207, E3 +321806.618}
SPL {X  -159.990, Y  +487.435, Z    +0.000, E1   +45.185, E3 +321818.910}
SPL {X  -159.990, Y  +477.648, Z    +0.000, E1   +46.080, E3 +321833.907}
SPL {X  -159.990, Y  +469.952, Z    +0.000, E1   +46.750, E3 +321845.415}
SPL {X  -159.990, Y  +460.762, Z    +0.000, E1   +47.755, E3 +321857.551}
SPL {X  -159.990, Y  +451.028, Z    +0.000, E1   +48.723, E3 +321870.163}
SPL {X  -159.990, Y  +441.023, Z    +0.000, E1   +49.655, E3 +321882.997}
SPL {X  -159.990, Y  +431.096, Z    +0.000, E1   +50.075, E3 +321898.285}
SPL {X  -159.990, Y  +423.834, Z    +0.000, E1   +50.037, E3 +321911.258}
SPL {X  -159.990, Y  +417.693, Z    +0.000, E1   +50.049, E3 +321922.156}
SPL {X  -159.990, Y  +408.922, Z    +0.000, E1   +50.085, E3 +321937.686}
SPL {X  -159.990, Y  +399.787, Z    +0.000, E1   +50.064, E3 +321953.955}
SPL {X  -159.990, Y  +393.038, Z    +0.000, E1   +50.038, E3 +321965.989}
SPL {X  -159.990, Y  +385.182, Z    +0.000, E1   +50.081, E3 +321979.906}
SPL {X  -159.906, Y  +377.302, Z    +0.000, E1   +50.024, E3 +321994.067}
SPL {X  -159.545, Y  +370.569, Z    +0.000, E1   +49.982, E3 +322006.380}
SPL {X  -158.871, Y  +363.614, Z    +0.000, E1   +49.855, E3 +322019.459}
SPL {X  -158.179, Y  +358.495, Z    +0.000, E1   +49.715, E3 +322029.308}
SPL {X  -157.354, Y  +353.576, Z    +0.000, E1   +49.583, E3 +322038.894}
SPL {X  -156.029, Y  +347.121, Z    +0.000, E1   +49.358, E3 +322051.711}
SPL {X  -154.686, Y  +341.646, Z    +0.000, E1   +49.094, E3 +322062.855}
SPL {X  -153.089, Y  +336.017, Z    +0.000, E1   +48.817, E3 +322074.464}
SPL {X  -151.481, Y  +331.019, Z    +0.000, E1   +48.491, E3 +322085.012}
SPL {X  -149.787, Y  +326.281, Z    +0.000, E1   +48.192, E3 +322095.100}
SPL {X  -148.124, Y  +322.035, Z    +0.000, E1   +47.846, E3 +322104.324}
SPL {X  -146.510, Y  +318.222, Z    +0.000, E1   +47.558, E3 +322112.636}
SPL {X  -141.189, Y  +307.250, Z    +0.000, E1   +40.067, E3 +322198.810}
ENDSPLINE

SPLINE
SPL {X  -154.923, Y  +342.556, Z    +0.000, E1   +23.930, E3 +322260.309}
SPL {X  -158.138, Y  +358.230, Z    +0.000, E1   +16.243, E3 +322269.267}
SPL {X  -159.647, Y  +372.034, Z    +0.000, E1    +8.739, E3 +322273.631}
SPL {X  -159.989, Y  +381.927, Z    +0.000, E1    +2.565, E3 +322275.391}
SPL {X  -159.990, Y  +386.909, Z    +0.000, E1    -1.211, E3 +322275.934}
SPL {X  -159.990, Y  +390.921, Z    +0.000, E1    -5.111, E3 +322276.413}
SPL {X  -159.990, Y  +395.719, Z    +0.000, E1   -10.396, E3 +322277.232}
SPL {X  -159.990, Y  +400.739, Z    +0.000, E1   -16.236, E3 +322278.430}
SPL {X  -159.990, Y  +409.482, Z    +0.000, E1   -25.418, E3 +322281.635}
SPL {X  -159.990, Y  +440.741, Z    +0.000, E1   -43.570, E3 +322302.292}
SPL {X  -159.990, Y  +488.072, Z    +0.000, E1   -48.834, E3 +322363.414}
SPL {X  -159.990, Y  +495.397, Z    +0.000, E1   -48.860, E3 +322376.963}
SPL {X  -159.990, Y  +502.531, Z    +0.000, E1   -48.834, E3 +322390.242}
SPL {X  -159.990, Y  +508.013, Z    +0.000, E1   -48.835, E3 +322400.377}
SPL {X  -159.990, Y  +513.813, Z    +0.000, E1   -48.843, E3 +322411.125}
SPL {X  -159.990, Y  +519.614, Z    +0.000, E1   -48.832, E3 +322421.926}
SPL {X  -159.990, Y  +524.730, Z    +0.000, E1   -48.830, E3 +322431.410}
SPL {X  -159.990, Y  +532.076, Z    +0.000, E1   -48.872, E3 +322444.975}
SPL {X  -159.990, Y  +539.248, Z    +0.000, E1   -48.832, E3 +322458.343}
SPL {X  -159.990, Y  +544.926, Z    +0.000, E1   -48.835, E3 +322468.872}
SPL {X  -159.990, Y  +550.252, Z    +0.000, E1   -48.827, E3 +322478.778}
SPL {X  -159.990, Y  +555.692, Z    +0.000, E1   -48.830, E3 +322488.875}
SPL {X  -159.990, Y  +561.308, Z    +0.000, E1   -48.827, E3 +322499.322}
SPL {X  -159.990, Y  +566.669, Z    +0.000, E1   -48.820, E3 +322509.271}
SPL {X  -159.990, Y  +572.248, Z    +0.000, E1   -48.830, E3 +322519.616}
SPL {X  -159.990, Y  +577.770, Z    +0.000, E1   -48.821, E3 +322529.863}
SPL {X  -159.990, Y  +583.108, Z    +0.000, E1   -48.828, E3 +322539.765}
SPL {X  -159.990, Y  +588.804, Z    +0.000, E1   -48.829, E3 +322550.322}
SPL {X  -159.990, Y  +594.280, Z    +0.000, E1   -48.826, E3 +322560.484}
SPL {X  -159.990, Y  +600.107, Z    +0.000, E1   -48.833, E3 +322571.298}
SPL {X  -159.990, Y  +605.910, Z    +0.000, E1   -48.823, E3 +322582.077}
SPL {X  -159.990, Y  +611.566, Z    +0.000, E1   -48.829, E3 +322592.566}
SPL {X  -159.990, Y  +617.357, Z    +0.000, E1   -48.824, E3 +322603.321}
SPL {X  -159.990, Y  +622.965, Z    +0.000, E1   -48.826, E3 +322613.720}
SPL {X  -159.990, Y  +629.255, Z    +0.000, E1   -48.834, E3 +322625.387}
SPL {X  -159.990, Y  +634.905, Z    +0.000, E1   -48.821, E3 +322635.884}
SPL {X  -159.990, Y  +640.372, Z    +0.000, E1   -48.828, E3 +322646.021}
SPL {X  -159.990, Y  +646.939, Z    +0.000, E1   -48.838, E3 +322658.191}
SPL {X  -159.990, Y  +653.448, Z    +0.000, E1   -48.827, E3 +322670.286}
SPL {X  -159.990, Y  +659.039, Z    +0.000, E1   -48.826, E3 +322680.650}
SPL {X  -159.990, Y  +664.817, Z    +0.000, E1   -48.832, E3 +322691.365}
SPL {X  -159.990, Y  +671.221, Z    +0.000, E1   -48.836, E3 +322703.238}
SPL {X  -159.887, Y  +677.230, Z    +0.000, E1   -48.811, E3 +322714.504}
SPL {X  -159.602, Y  +682.629, Z    +0.000, E1   -48.761, E3 +322724.837}
SPL {X  -159.150, Y  +687.876, Z    +0.000, E1   -48.673, E3 +322735.076}
SPL {X  -158.569, Y  +692.776, Z    +0.000, E1   -48.570, E3 +322744.784}
SPL {X  -157.870, Y  +697.458, Z    +0.000, E1   -48.439, E3 +322754.213}
SPL {X  -157.028, Y  +702.144, Z    +0.000, E1   -48.297, E3 +322763.761}
SPL {X  -155.977, Y  +707.110, Z    +0.000, E1   -48.106, E3 +322774.065}
SPL {X  -154.657, Y  +712.464, Z    +0.000, E1   -47.874, E3 +322785.349}
SPL {X  -153.406, Y  +716.924, Z    +0.000, E1   -47.628, E3 +322794.915}
SPL {X  -152.020, Y  +721.367, Z    +0.000, E1   -47.374, E3 +322804.566}
SPL {X  -150.440, Y  +725.947, Z    +0.000, E1   -47.070, E3 +322814.671}
SPL {X  -148.730, Y  +730.459, Z    +0.000, E1   -46.749, E3 +322824.722}
SPL {X  -147.178, Y  +734.233, Z    +0.000, E1   -46.439, E3 +322833.256}
SPL {X  -140.263, Y  +748.461, Z    +0.000, E1   -42.675, E3 +322891.594}
ENDSPLINE

SPLINE
SPL {X  -141.835, Y  +745.525, Z    +0.000, E1   -39.068, E3 +322923.595}
SPL {X  -152.406, Y  +720.176, Z    +0.000, E1   -27.814, E3 +322974.808}
SPL {X  -157.542, Y  +699.382, Z    +0.000, E1   -18.086, E3 +322989.141}
SPL {X  -159.386, Y  +685.393, Z    +0.000, E1   -10.664, E3 +322994.095}
SPL {X  -159.928, Y  +675.946, Z    +0.000, E1    -5.007, E3 +322996.134}
SPL {X  -159.990, Y  +671.468, Z    +0.000, E1    -2.030, E3 +322996.730}
SPL {X  -159.990, Y  +667.678, Z    +0.000, E1    +0.783, E3 +322997.080}
SPL {X  -159.990, Y  +663.139, Z    +0.000, E1    +5.135, E3 +322997.597}
SPL {X  -159.990, Y  +658.551, Z    +0.000, E1   +10.313, E3 +322998.371}
SPL {X  -159.990, Y  +653.526, Z    +0.000, E1   +16.156, E3 +322999.606}
SPL {X  -159.990, Y  +644.434, Z    +0.000, E1   +25.921, E3 +323002.801}
SPL {X  -159.990, Y  +612.255, Z    +0.000, E1   +44.102, E3 +323024.682}
SPL {X  -159.990, Y  +561.053, Z    +0.000, E1   +49.668, E3 +323089.515}
SPL {X  -159.990, Y  +552.984, Z    +0.000, E1   +49.619, E3 +323104.156}
SPL {X  -159.990, Y  +547.278, Z    +0.000, E1   +49.619, E3 +323114.455}
SPL {X  -159.990, Y  +538.738, Z    +0.000, E1   +49.672, E3 +323129.779}
SPL {X  -159.990, Y  +529.436, Z    +0.000, E1   +49.638, E3 +323146.603}
SPL {X  -159.990, Y  +522.804, Z    +0.000, E1   +49.620, E3 +323158.592}
SPL {X  -159.990, Y  +515.173, Z    +0.000, E1   +49.653, E3 +323172.330}
SPL {X  -159.990, Y  +505.896, Z    +0.000, E1   +49.645, E3 +323189.105}
SPL {X  -159.990, Y  +503.881, Z    +0.000, E1   +48.376, E3 +323200.092}
ENDSPLINE

SPLINE
SPL {X  -159.990, Y  +518.841, Z    +0.000, E1   +41.643, E3 +323209.543}
ENDSPLINE

SPLINE
SPL {X  -159.990, Y  +508.096, Z    +0.000, E1   +42.952, E3 +323226.810}
SPL {X  -159.990, Y  +500.642, Z    +0.000, E1   +43.747, E3 +323238.731}
SPL {X  -159.990, Y  +492.511, Z    +0.000, E1   +44.632, E3 +323251.383}
SPL {X  -159.990, Y  +482.131, Z    +0.000, E1   +45.680, E3 +323267.053}
SPL {X  -159.990, Y  +472.111, Z    +0.000, E1   +46.581, E3 +323282.185}
SPL {X  -159.990, Y  +462.892, Z    +0.000, E1   +47.497, E3 +323294.899}
SPL {X  -159.990, Y  +452.841, Z    +0.000, E1   +48.572, E3 +323307.746}
SPL {X  -159.990, Y  +441.023, Z    +0.000, E1   +49.655, E3 +323322.997}
SPL {X  -159.990, Y  +431.096, Z    +0.000, E1   +50.075, E3 +323338.285}
SPL {X  -159.990, Y  +423.834, Z    +0.000, E1   +50.037, E3 +323351.258}
SPL {X  -159.990, Y  +417.693, Z    +0.000, E1   +50.049, E3 +323362.156}
SPL {X  -159.990, Y  +411.447, Z    +0.000, E1   +50.039, E3 +323373.275}
SPL {X  -159.990, Y  +406.170, Z    +0.000, E1   +50.036, E3 +323382.647}
SPL {X  -159.990, Y  +399.787, Z    +0.000, E1   +50.064, E3 +323393.955}
SPL {X  -159.990, Y  +393.038, Z    +0.000, E1   +50.038, E3 +323405.989}
SPL {X  -159.990, Y  +385.182, Z    +0.000, E1   +50.081, E3 +323419.906}
SPL {X  -159.906, Y  +377.302, Z    +0.000, E1   +50.024, E3 +323434.067}
SPL {X  -159.545, Y  +370.569, Z    +0.000, E1   +49.982, E3 +323446.380}
SPL {X  -158.871, Y  +363.614, Z    +0.000, E1   +49.855, E3 +323459.459}
SPL {X  -158.179, Y  +358.495, Z    +0.000, E1   +49.715, E3 +323469.308}
SPL {X  -157.354, Y  +353.576, Z    +0.000, E1   +49.583, E3 +323478.894}
SPL {X  -156.029, Y  +347.121, Z    +0.000, E1   +49.358, E3 +323491.711}
SPL {X  -154.686, Y  +341.646, Z    +0.000, E1   +49.094, E3 +323502.855}
SPL {X  -153.439, Y  +337.188, Z    +0.000, E1   +48.857, E3 +323512.062}
SPL {X  -151.836, Y  +332.074, Z    +0.000, E1   +48.585, E3 +323522.738}
SPL {X  -150.221, Y  +327.451, Z    +0.000, E1   +48.251, E3 +323532.616}
SPL {X  -148.587, Y  +323.181, Z    +0.000, E1   +47.960, E3 +323541.800}
SPL {X  -146.510, Y  +318.222, Z    +0.000, E1   +47.558, E3 +323552.636}
SPL {X  -141.189, Y  +307.250, Z    +0.000, E1   +40.067, E3 +323638.810}
ENDSPLINE

